LIN {X 0,Y 467.594,Z 791.05,A -85,B 0,C 180,E1 -7505.746,E2 -7505.746} C_VEL
LIN {X 0,Y 467.216,Z 798.675,A -85,B 0,C 180,E1 -7507.133,E2 -7507.133} C_VEL
LIN {X 0,Y 467.007,Z 804.577,A -85,B 0,C 180,E1 -7508.506,E2 -7508.506} C_VEL
LIN {X 0,Y 466.843,Z 809.072,A -85,B 0,C 180,E1 -7509.847,E2 -7509.847} C_VEL
LIN {X 0,Y 466.705,Z 813.073,A -85,B 0,C 180,E1 -7511.496,E2 -7511.496} C_VEL
LIN {X 0,Y 466.63,Z 814.936,A -85,B 0,C 180,E1 -7512.667,E2 -7512.667} C_VEL
LIN {X 0,Y 466.577,Z 816.084,A -85,B 0,C 180,E1 -7513.858,E2 -7513.858} C_VEL
LIN {X 0,Y 466.568,Z 816.491,A -85,B 0,C 180,E1 -7515.069,E2 -7515.069} C_VEL
LIN {X 0,Y 466.584,Z 816.072,A -85,B 0,C 180,E1 -7516.302,E2 -7516.302} C_VEL
LIN {X 0,Y 466.641,Z 814.812,A -85,B 0,C 180,E1 -7517.558,E2 -7517.558} C_VEL
LIN {X 0,Y 466.745,Z 812.646,A -85,B 0,C 180,E1 -7518.838,E2 -7518.838} C_VEL
LIN {X 0,Y 466.842,Z 809.444,A -85,B 0,C 180,E1 -7520.152,E2 -7520.152} C_VEL
LIN {X 0,Y 467.011,Z 805.061,A -85,B 0,C 180,E1 -7521.492,E2 -7521.492} C_VEL
LIN {X 0,Y 467.267,Z 798.57,A -85,B 0,C 180,E1 -7523.014,E2 -7523.014} C_VEL
LIN {X 0,Y 467.568,Z 791.804,A -85,B 0,C 180,E1 -7524.258,E2 -7524.258} C_VEL
LIN {X 0,Y 467.987,Z 783.664,A -85,B 0,C 180,E1 -7525.471,E2 -7525.471} C_VEL
LIN {X 0,Y 468.465,Z 774.171,A -85,B 0,C 180,E1 -7526.621,E2 -7526.621} C_VEL
LIN {X 0,Y 468.906,Z 764.185,A -85,B 0,C 180,E1 -7527.601,E2 -7527.601} C_VEL
LIN {X 0,Y 469.422,Z 752.274,A -85,B 0,C 180,E1 -7528.524,E2 -7528.524} C_VEL
LIN {X 0,Y 469.902,Z 740.221,A -85,B 0,C 180,E1 -7529.249,E2 -7529.249} C_VEL
LIN {X 0,Y 470.237,Z 727.327,A -85,B 0,C 180,E1 -7529.816,E2 -7529.816} C_VEL
LIN {X 0,Y 470.482,Z 714.641,A -85,B 0,C 180,E1 -7530.195,E2 -7530.195} C_VEL
LIN {X 0,Y 470.92,Z 673.673,A -85,B 0,C 180,E1 -7530.864,E2 -7530.864} C_VEL
LIN {X 0,Y 471.328,Z 620.727,A -85,B 0,C 180,E1 -7531.703,E2 -7531.703} C_VEL
LIN {X 0,Y 468.51,Z 607.159,A -85,B 0,C 180,E1 -7532.05,E2 -7532.05} C_VEL
LIN {X 0,Y 468.72,Z 598.189,A -85,B 0,C 180,E1 -7534.108,E2 -7534.108} C_VEL
LIN {X 0,Y 467.618,Z 592.238,A -85,B 0,C 180,E1 -7535.588,E2 -7535.588} C_VEL
LIN {X 0,Y 467.576,Z 592.244,A -85,B 0,C 180,E1 -7538.855,E2 -7538.855} C_VEL
LIN {X 0,Y 467.622,Z 592.234,A -85,B 0,C 180,E1 -7541.603,E2 -7541.603} C_VEL
LIN {X 0,Y 467.628,Z 592.236,A -85,B 0,C 180,E1 -7544.305,E2 -7544.305} C_VEL
LIN {X 0,Y 467.687,Z 592.225,A -85,B 0,C 180,E1 -7547.856,E2 -7547.856} C_VEL
LIN {X 0,Y 467.673,Z 592.229,A -85,B 0,C 180,E1 -7551.358,E2 -7551.358} C_VEL
LIN {X 0,Y 467.744,Z 592.218,A -85,B 0,C 180,E1 -7553.963,E2 -7553.963} C_VEL
LIN {X 0,Y 467.858,Z 592.205,A -85,B 0,C 180,E1 -7557.418,E2 -7557.418} C_VEL
LIN {X 0,Y 467.872,Z 592.201,A -85,B 0,C 180,E1 -7560,E2 -7560} C_VEL
LIN {X 0,Y 467.852,Z 592.207,A -85,B 0,C 180,E1 -7562.583,E2 -7562.583} C_VEL
LIN {X 0,Y 467.745,Z 592.216,A -85,B 0,C 180,E1 -7566.038,E2 -7566.038} C_VEL
LIN {X 0,Y 467.674,Z 592.23,A -85,B 0,C 180,E1 -7568.643,E2 -7568.643} C_VEL
LIN {X 0,Y 467.673,Z 592.225,A -85,B 0,C 180,E1 -7572.145,E2 -7572.145} C_VEL
LIN {X 0,Y 467.64,Z 592.227,A -85,B 0,C 180,E1 -7575.886,E2 -7575.886} C_VEL
LIN {X 0,Y 467.616,Z 592.237,A -85,B 0,C 180,E1 -7579.308,E2 -7579.308} C_VEL
LIN {X 0,Y 467.526,Z 592.242,A -85,B 0,C 180,E1 -7582.075,E2 -7582.075} C_VEL
LIN {X 0,Y 467.596,Z 592.239,A -85,B 0,C 180,E1 -7584.888,E2 -7584.888} C_VEL
LIN {X 0,Y 467.622,Z 592.232,A -85,B 0,C 180,E1 -7587.769,E2 -7587.769} C_VEL
LIN {X 0,Y 467.573,Z 592.242,A -85,B 0,C 180,E1 -7591.048,E2 -7591.048} C_VEL
LIN {X 0,Y 467.584,Z 592.235,A -85,B 0,C 180,E1 -7594.244,E2 -7594.244} C_VEL
LIN {X 0,Y 467.547,Z 592.247,A -85,B 0,C 180,E1 -7597.188,E2 -7597.188} C_VEL
LIN {X 0,Y 467.579,Z 592.236,A -85,B 0,C 180,E1 -7600.265,E2 -7600.265} C_VEL
LIN {X 0,Y 467.582,Z 592.238,A -85,B 0,C 180,E1 -7602.568,E2 -7602.568} C_VEL
LIN {X 0,Y 467.567,Z 592.243,A -85,B 0,C 180,E1 -7605.054,E2 -7605.054} C_VEL
LIN {X 0,Y 467.586,Z 592.244,A -85,B 0,C 180,E1 -7607.441,E2 -7607.441} C_VEL
LIN {X 0,Y 467.613,Z 592.235,A -85,B 0,C 180,E1 -7610.86,E2 -7610.86} C_VEL
LIN {X 0,Y 467.562,Z 592.242,A -85,B 0,C 180,E1 -7614.261,E2 -7614.261} C_VEL
LIN {X 0,Y 467.581,Z 592.244,A -85,B 0,C 180,E1 -7617.322,E2 -7617.322} C_VEL
LIN {X 0,Y 467.57,Z 592.242,A -85,B 0,C 180,E1 -7620.668,E2 -7620.668} C_VEL
LIN {X 0,Y 467.68,Z 592.255,A -85,B 0,C 180,E1 -7623.265,E2 -7623.265} C_VEL
LIN {X 0,Y 470.039,Z 604.523,A -85,B 0,C 180,E1 -7625.573,E2 -7625.573} C_VEL
LIN {X 0,Y 469.976,Z 610.728,A -85,B 0,C 180,E1 -7626.655,E2 -7626.655} C_VEL
LIN {X 0,Y 469.08,Z 629.475,A -85,B 0,C 180,E1 -7629.843,E2 -7629.843} C_VEL
LIN {X 0,Y 468.442,Z 645.546,A -85,B 0,C 180,E1 -7632.539,E2 -7632.539} C_VEL
LIN {X 0,Y 468.36,Z 648.312,A -85,B 0,C 180,E1 -7632.979,E2 -7632.979} C_VEL
LIN {X 0,Y 471.137,Z 667.101,A -85,B 0,C 180,E1 -7633.385,E2 -7633.385} C_VEL
LIN {X 0,Y 470.407,Z 757.136,A -85,B 0,C 180,E1 -7634.816,E2 -7634.816} C_VEL
LIN {X 0,Y 470.035,Z 770.301,A -85,B 0,C 180,E1 -7635.192,E2 -7635.192} C_VEL
LIN {X 0,Y 469.668,Z 782.454,A -85,B 0,C 180,E1 -7635.706,E2 -7635.706} C_VEL
LIN {X 0,Y 469.19,Z 793.935,A -85,B 0,C 180,E1 -7636.355,E2 -7636.355} C_VEL
LIN {X 0,Y 468.694,Z 805.881,A -85,B 0,C 180,E1 -7637.234,E2 -7637.234} C_VEL
LIN {X 0,Y 468.248,Z 816.36,A -85,B 0,C 180,E1 -7638.2,E2 -7638.2} C_VEL
LIN {X 0,Y 467.768,Z 825.036,A -85,B 0,C 180,E1 -7639.175,E2 -7639.175} C_VEL
LIN {X 0,Y 467.427,Z 833.045,A -85,B 0,C 180,E1 -7640.262,E2 -7640.262} C_VEL
LIN {X 0,Y 467.126,Z 840.876,A -85,B 0,C 180,E1 -7641.565,E2 -7641.565} C_VEL
LIN {X 0,Y 466.855,Z 848.078,A -85,B 0,C 180,E1 -7643.083,E2 -7643.083} C_VEL
LIN {X 0,Y 466.787,Z 852.882,A -85,B 0,C 180,E1 -7644.384,E2 -7644.384} C_VEL
LIN {X 0,Y 466.662,Z 856.552,A -85,B 0,C 180,E1 -7645.682,E2 -7645.682} C_VEL
LIN {X 0,Y 466.727,Z 858.454,A -85,B 0,C 180,E1 -7646.547,E2 -7646.547} C_VEL
LIN {X 0,Y 466.681,Z 859.877,A -85,B 0,C 180,E1 -7647.411,E2 -7647.411} C_VEL
LIN {X 0,Y 466.661,Z 860.895,A -85,B 0,C 180,E1 -7648.274,E2 -7648.274} C_VEL
LIN {X 0,Y 466.62,Z 861.518,A -85,B 0,C 180,E1 -7649.137,E2 -7649.137} C_VEL
LIN {X 0,Y 466.598,Z 861.745,A -85,B 0,C 180,E1 -7650,E2 -7650} C_VEL
LIN {X 0,Y 466.62,Z 861.534,A -85,B 0,C 180,E1 -7650.863,E2 -7650.863} C_VEL
LIN {X 0,Y 466.661,Z 860.929,A -85,B 0,C 180,E1 -7651.726,E2 -7651.726} C_VEL
LIN {X 0,Y 466.68,Z 859.93,A -85,B 0,C 180,E1 -7652.589,E2 -7652.589} C_VEL
LIN {X 0,Y 466.696,Z 858.521,A -85,B 0,C 180,E1 -7653.453,E2 -7653.453} C_VEL
LIN {X 0,Y 466.7,Z 855.559,A -85,B 0,C 180,E1 -7654.751,E2 -7654.751} C_VEL
LIN {X 0,Y 466.773,Z 851.546,A -85,B 0,C 180,E1 -7656.05,E2 -7656.05} C_VEL
LIN {X 0,Y 466.946,Z 845.366,A -85,B 0,C 180,E1 -7657.567,E2 -7657.567} C_VEL
LIN {X 0,Y 467.2,Z 838.62,A -85,B 0,C 180,E1 -7658.87,E2 -7658.87} C_VEL
LIN {X 0,Y 467.526,Z 830.248,A -85,B 0,C 180,E1 -7660.173,E2 -7660.173} C_VEL
LIN {X 0,Y 467.953,Z 821.64,A -85,B 0,C 180,E1 -7661.259,E2 -7661.259} C_VEL
LIN {X 0,Y 468.462,Z 811.469,A -85,B 0,C 180,E1 -7662.302,E2 -7662.302} C_VEL
LIN {X 0,Y 468.896,Z 800.495,A -85,B 0,C 180,E1 -7663.213,E2 -7663.213} C_VEL
LIN {X 0,Y 469.425,Z 788.908,A -85,B 0,C 180,E1 -7663.97,E2 -7663.97} C_VEL
LIN {X 0,Y 469.859,Z 776.886,A -85,B 0,C 180,E1 -7664.564,E2 -7664.564} C_VEL
LIN {X 0,Y 470.29,Z 763.907,A -85,B 0,C 180,E1 -7665.021,E2 -7665.021} C_VEL
LIN {X 0,Y 470.563,Z 750.082,A -85,B 0,C 180,E1 -7665.317,E2 -7665.317} C_VEL
LIN {X 0,Y 471.142,Z 667.137,A -85,B 0,C 180,E1 -7666.617,E2 -7666.617} C_VEL
LIN {X 0,Y 468.397,Z 648.688,A -85,B 0,C 180,E1 -7667.026,E2 -7667.026} C_VEL
LIN {X 0,Y 469.166,Z 630.051,A -85,B 0,C 180,E1 -7670.153,E2 -7670.153} C_VEL
LIN {X 0,Y 469.917,Z 613.979,A -85,B 0,C 180,E1 -7672.882,E2 -7672.882} C_VEL
LIN {X 0,Y 470.161,Z 604.995,A -85,B 0,C 180,E1 -7674.438,E2 -7674.438} C_VEL
LIN {X 0,Y 467.687,Z 592.23,A -85,B 0,C 180,E1 -7676.851,E2 -7676.851} C_VEL
LIN {X 0,Y 467.554,Z 592.244,A -85,B 0,C 180,E1 -7679.737,E2 -7679.737} C_VEL
LIN {X 0,Y 467.583,Z 592.241,A -85,B 0,C 180,E1 -7682.757,E2 -7682.757} C_VEL
LIN {X 0,Y 467.556,Z 592.24,A -85,B 0,C 180,E1 -7685.888,E2 -7685.888} C_VEL
LIN {X 0,Y 467.598,Z 592.235,A -85,B 0,C 180,E1 -7689.142,E2 -7689.142} C_VEL
LIN {X 0,Y 467.584,Z 592.244,A -85,B 0,C 180,E1 -7692.566,E2 -7692.566} C_VEL
LIN {X 0,Y 467.567,Z 592.241,A -85,B 0,C 180,E1 -7695.052,E2 -7695.052} C_VEL
LIN {X 0,Y 467.585,Z 592.236,A -85,B 0,C 180,E1 -7697.439,E2 -7697.439} C_VEL
LIN {X 0,Y 467.588,Z 592.242,A -85,B 0,C 180,E1 -7700.855,E2 -7700.855} C_VEL
LIN {X 0,Y 467.558,Z 592.241,A -85,B 0,C 180,E1 -7704.259,E2 -7704.259} C_VEL
LIN {X 0,Y 467.576,Z 592.239,A -85,B 0,C 180,E1 -7707.32,E2 -7707.32} C_VEL
LIN {X 0,Y 467.572,Z 592.242,A -85,B 0,C 180,E1 -7710.664,E2 -7710.664} C_VEL
LIN {X 0,Y 467.621,Z 592.236,A -85,B 0,C 180,E1 -7713.2,E2 -7713.2} C_VEL
LIN {X 0,Y 467.585,Z 592.237,A -85,B 0,C 180,E1 -7716.467,E2 -7716.467} C_VEL
LIN {X 0,Y 467.616,Z 592.232,A -85,B 0,C 180,E1 -7719.776,E2 -7719.776} C_VEL
LIN {X 0,Y 467.6,Z 592.235,A -85,B 0,C 180,E1 -7722.506,E2 -7722.506} C_VEL
LIN {X 0,Y 467.598,Z 592.243,A -85,B 0,C 180,E1 -7725.196,E2 -7725.196} C_VEL
LIN {X 0,Y 467.647,Z 592.229,A -85,B 0,C 180,E1 -7727.854,E2 -7727.854} C_VEL
LIN {X 0,Y 467.673,Z 592.232,A -85,B 0,C 180,E1 -7731.357,E2 -7731.357} C_VEL
LIN {X 0,Y 467.739,Z 592.217,A -85,B 0,C 180,E1 -7733.962,E2 -7733.962} C_VEL
LIN {X 0,Y 467.851,Z 592.211,A -85,B 0,C 180,E1 -7737.417,E2 -7737.417} C_VEL
LIN {X 0,Y 467.872,Z 592.201,A -85,B 0,C 180,E1 -7740,E2 -7740} C_VEL
LIN {X 0,Y 467.851,Z 592.202,A -85,B 0,C 180,E1 -7742.582,E2 -7742.582} C_VEL
LIN {X 0,Y 467.742,Z 592.218,A -85,B 0,C 180,E1 -7746.037,E2 -7746.037} C_VEL
LIN {X 0,Y 467.672,Z 592.224,A -85,B 0,C 180,E1 -7748.642,E2 -7748.642} C_VEL
LIN {X 0,Y 467.646,Z 592.23,A -85,B 0,C 180,E1 -7752.145,E2 -7752.145} C_VEL
LIN {X 0,Y 467.628,Z 592.238,A -85,B 0,C 180,E1 -7755.695,E2 -7755.695} C_VEL
LIN {X 0,Y 467.607,Z 592.233,A -85,B 0,C 180,E1 -7758.765,E2 -7758.765} C_VEL
LIN {X 0,Y 467.57,Z 592.239,A -85,B 0,C 180,E1 -7761.268,E2 -7761.268} C_VEL
LIN {X 0,Y 467.563,Z 592.246,A -85,B 0,C 180,E1 -7763.943,E2 -7763.943} C_VEL
LIN {X 0,Y 467.617,Z 592.231,A -85,B 0,C 180,E1 -7766.8,E2 -7766.8} C_VEL
LIN {X 0,Y 467.577,Z 592.241,A -85,B 0,C 180,E1 -7769.736,E2 -7769.736} C_VEL
LIN {X 0,Y 467.574,Z 592.237,A -85,B 0,C 180,E1 -7772.758,E2 -7772.758} C_VEL
LIN {X 0,Y 467.547,Z 592.246,A -85,B 0,C 180,E1 -7775.89,E2 -7775.89} C_VEL
LIN {X 0,Y 467.615,Z 592.232,A -85,B 0,C 180,E1 -7779.141,E2 -7779.141} C_VEL
LIN {X 0,Y 467.611,Z 592.236,A -85,B 0,C 180,E1 -7782.572,E2 -7782.572} C_VEL
LIN {X 0,Y 467.559,Z 592.246,A -85,B 0,C 180,E1 -7786.178,E2 -7786.178} C_VEL
LIN {X 0,Y 467.574,Z 592.24,A -85,B 0,C 180,E1 -7788.723,E2 -7788.723} C_VEL
LIN {X 0,Y 467.559,Z 592.241,A -85,B 0,C 180,E1 -7791.956,E2 -7791.956} C_VEL
LIN {X 0,Y 467.562,Z 592.239,A -85,B 0,C 180,E1 -7795.168,E2 -7795.168} C_VEL
LIN {X 0,Y 467.578,Z 592.241,A -85,B 0,C 180,E1 -7798.26,E2 -7798.26} C_VEL
LIN {X 0,Y 467.571,Z 592.238,A -85,B 0,C 180,E1 -7801.251,E2 -7801.251} C_VEL
LIN {X 0,Y 467.611,Z 592.234,A -85,B 0,C 180,E1 -7803.2,E2 -7803.2} C_VEL
LIN {X 0,Y 467.588,Z 592.241,A -85,B 0,C 180,E1 -7806.468,E2 -7806.468} C_VEL
LIN {X 0,Y 467.62,Z 592.231,A -85,B 0,C 180,E1 -7809.778,E2 -7809.778} C_VEL
LIN {X 0,Y 467.606,Z 592.238,A -85,B 0,C 180,E1 -7812.507,E2 -7812.507} C_VEL
LIN {X 0,Y 467.595,Z 592.235,A -85,B 0,C 180,E1 -7815.433,E2 -7815.433} C_VEL
LIN {X 0,Y 466.928,Z 592.319,A -85,B 0,C 180,E1 -7816.152,E2 -7816.152} C_VEL
LIN {X 0,Y 464.084,Z 592.674,A -85,B 0,C 180,E1 -7817.32,E2 -7817.32} C_VEL
LIN {X 0,Y 461.682,Z 592.972,A -85,B 0,C 180,E1 -7818.262,E2 -7818.262} C_VEL
LIN {X 0,Y 460.655,Z 593.106,A -85,B 0,C 180,E1 -7818.99,E2 -7818.99} C_VEL
LIN {X 0,Y 460.574,Z 593.11,A -85,B 0,C 180,E1 -7819.236,E2 -7819.236} C_VEL
LIN {X 0,Y 460.712,Z 593.095,A -85,B 0,C 180,E1 -7822.543,E2 -7822.543} C_VEL
LIN {X 0,Y 460.692,Z 593.099,A -85,B 0,C 180,E1 -7824.748,E2 -7824.748} C_VEL
LIN {X 0,Y 460.822,Z 593.082,A -85,B 0,C 180,E1 -7827.378,E2 -7827.378} C_VEL
LIN {X 0,Y 460.851,Z 593.074,A -85,B 0,C 180,E1 -7830,E2 -7830} C_VEL
LIN {X 0,Y 460.823,Z 593.08,A -85,B 0,C 180,E1 -7832.622,E2 -7832.622} C_VEL
LIN {X 0,Y 460.698,Z 593.093,A -85,B 0,C 180,E1 -7836.13,E2 -7836.13} C_VEL
LIN {X 0,Y 460.625,Z 593.105,A -85,B 0,C 180,E1 -7838.776,E2 -7838.776} C_VEL
LIN {X 0,Y 460.61,Z 593.104,A -85,B 0,C 180,E1 -7842.445,E2 -7842.445} C_VEL
LIN {X 0,Y 460.596,Z 593.107,A -85,B 0,C 180,E1 -7845.997,E2 -7845.997} C_VEL
LIN {X 0,Y 460.567,Z 593.112,A -85,B 0,C 180,E1 -7848.902,E2 -7848.902} C_VEL
LIN {X 0,Y 460.512,Z 593.125,A -85,B 0,C 180,E1 -7851.485,E2 -7851.485} C_VEL
LIN {X 0,Y 460.633,Z 593.212,A -85,B 0,C 180,E1 -7854.627,E2 -7854.627} C_VEL
LIN {X 0,Y 461.71,Z 599.757,A -85,B 0,C 180,E1 -7856.194,E2 -7856.194} C_VEL
LIN {X 0,Y 461.51,Z 606.979,A -85,B 0,C 180,E1 -7857.811,E2 -7857.811} C_VEL
LIN {X 0,Y 464.568,Z 622.378,A -85,B 0,C 180,E1 -7858.182,E2 -7858.182} C_VEL
LIN {X 0,Y 463.656,Z 713.559,A -85,B 0,C 180,E1 -7859.653,E2 -7859.653} C_VEL
LIN {X 0,Y 463.357,Z 727.425,A -85,B 0,C 180,E1 -7860.067,E2 -7860.067} C_VEL
LIN {X 0,Y 462.965,Z 740.325,A -85,B 0,C 180,E1 -7860.643,E2 -7860.643} C_VEL
LIN {X 0,Y 462.477,Z 752.601,A -85,B 0,C 180,E1 -7861.394,E2 -7861.394} C_VEL
LIN {X 0,Y 461.936,Z 764.155,A -85,B 0,C 180,E1 -7862.302,E2 -7862.302} C_VEL
LIN {X 0,Y 461.425,Z 774.936,A -85,B 0,C 180,E1 -7863.381,E2 -7863.381} C_VEL
LIN {X 0,Y 460.939,Z 784.574,A -85,B 0,C 180,E1 -7864.58,E2 -7864.58} C_VEL
LIN {X 0,Y 460.564,Z 792.034,A -85,B 0,C 180,E1 -7865.717,E2 -7865.717} C_VEL
LIN {X 0,Y 460.156,Z 799.828,A -85,B 0,C 180,E1 -7867.199,E2 -7867.199} C_VEL
LIN {X 0,Y 459.908,Z 806.333,A -85,B 0,C 180,E1 -7868.8,E2 -7868.8} C_VEL
LIN {X 0,Y 459.725,Z 810.475,A -85,B 0,C 180,E1 -7870.15,E2 -7870.15} C_VEL
LIN {X 0,Y 459.618,Z 813.471,A -85,B 0,C 180,E1 -7871.475,E2 -7871.475} C_VEL
LIN {X 0,Y 459.547,Z 815.452,A -85,B 0,C 180,E1 -7872.771,E2 -7872.771} C_VEL
LIN {X 0,Y 459.479,Z 816.535,A -85,B 0,C 180,E1 -7874.038,E2 -7874.038} C_VEL
LIN {X 0,Y 459.472,Z 816.802,A -85,B 0,C 180,E1 -7875.284,E2 -7875.284} C_VEL
LIN {X 0,Y 459.511,Z 816.299,A -85,B 0,C 180,E1 -7876.509,E2 -7876.509} C_VEL
LIN {X 0,Y 459.558,Z 815.019,A -85,B 0,C 180,E1 -7877.71,E2 -7877.71} C_VEL
LIN {X 0,Y 459.662,Z 813,A -85,B 0,C 180,E1 -7878.895,E2 -7878.895} C_VEL
LIN {X 0,Y 459.771,Z 810.274,A -85,B 0,C 180,E1 -7880.059,E2 -7880.059} C_VEL
LIN {X 0,Y 459.937,Z 805.782,A -85,B 0,C 180,E1 -7881.489,E2 -7881.489} C_VEL
LIN {X 0,Y 460.213,Z 799.458,A -85,B 0,C 180,E1 -7883.02,E2 -7883.02} C_VEL
LIN {X 0,Y 460.54,Z 792.863,A -85,B 0,C 180,E1 -7884.279,E2 -7884.279} C_VEL
LIN {X 0,Y 460.927,Z 785.531,A -85,B 0,C 180,E1 -7885.421,E2 -7885.421} C_VEL
LIN {X 0,Y 461.454,Z 776.05,A -85,B 0,C 180,E1 -7886.621,E2 -7886.621} C_VEL
LIN {X 0,Y 461.93,Z 765.542,A -85,B 0,C 180,E1 -7887.697,E2 -7887.697} C_VEL
LIN {X 0,Y 462.449,Z 754.398,A -85,B 0,C 180,E1 -7888.602,E2 -7888.602} C_VEL
LIN {X 0,Y 462.933,Z 742.386,A -85,B 0,C 180,E1 -7889.361,E2 -7889.361} C_VEL
LIN {X 0,Y 463.364,Z 729.575,A -85,B 0,C 180,E1 -7889.966,E2 -7889.966} C_VEL
LIN {X 0,Y 463.616,Z 716.872,A -85,B 0,C 180,E1 -7890.375,E2 -7890.375} C_VEL
LIN {X 0,Y 463.875,Z 697.07,A -85,B 0,C 180,E1 -7890.736,E2 -7890.736} C_VEL
LIN {X 0,Y 464.612,Z 621.891,A -85,B 0,C 180,E1 -7891.944,E2 -7891.944} C_VEL
LIN {X 0,Y 461.594,Z 607.587,A -85,B 0,C 180,E1 -7892.305,E2 -7892.305} C_VEL
LIN {X 0,Y 461.862,Z 600.852,A -85,B 0,C 180,E1 -7893.865,E2 -7893.865} C_VEL
LIN {X 0,Y 461.013,Z 595.306,A -85,B 0,C 180,E1 -7895.215,E2 -7895.215} C_VEL
LIN {X 0,Y 460.568,Z 593.117,A -85,B 0,C 180,E1 -7895.806,E2 -7895.806} C_VEL
LIN {X 0,Y 460.541,Z 593.116,A -85,B 0,C 180,E1 -7899.453,E2 -7899.453} C_VEL
LIN {X 0,Y 460.549,Z 593.118,A -85,B 0,C 180,E1 -7902.23,E2 -7902.23} C_VEL
LIN {X 0,Y 460.555,Z 593.118,A -85,B 0,C 180,E1 -7904.965,E2 -7904.965} C_VEL
LIN {X 0,Y 460.647,Z 593.102,A -85,B 0,C 180,E1 -7907.667,E2 -7907.667} C_VEL
LIN {X 0,Y 460.62,Z 593.108,A -85,B 0,C 180,E1 -7911.224,E2 -7911.224} C_VEL
LIN {X 0,Y 460.708,Z 593.094,A -85,B 0,C 180,E1 -7913.871,E2 -7913.871} C_VEL
LIN {X 0,Y 460.824,Z 593.081,A -85,B 0,C 180,E1 -7917.378,E2 -7917.378} C_VEL
LIN {X 0,Y 460.843,Z 593.077,A -85,B 0,C 180,E1 -7920,E2 -7920} C_VEL
LIN {X 0,Y 460.817,Z 593.084,A -85,B 0,C 180,E1 -7922.623,E2 -7922.623} C_VEL
LIN {X 0,Y 460.709,Z 593.093,A -85,B 0,C 180,E1 -7926.13,E2 -7926.13} C_VEL
LIN {X 0,Y 460.621,Z 593.11,A -85,B 0,C 180,E1 -7928.777,E2 -7928.777} C_VEL
LIN {X 0,Y 460.625,Z 593.105,A -85,B 0,C 180,E1 -7932.457,E2 -7932.457} C_VEL
LIN {X 0,Y 460.591,Z 593.105,A -85,B 0,C 180,E1 -7935.998,E2 -7935.998} C_VEL
LIN {X 0,Y 460.563,Z 593.116,A -85,B 0,C 180,E1 -7938.903,E2 -7938.903} C_VEL
LIN {X 0,Y 460.508,Z 593.12,A -85,B 0,C 180,E1 -7941.486,E2 -7941.486} C_VEL
LIN {X 0,Y 460.535,Z 593.115,A -85,B 0,C 180,E1 -7944.333,E2 -7944.333} C_VEL
LIN {X 0,Y 460.578,Z 593.116,A -85,B 0,C 180,E1 -7947.244,E2 -7947.244} C_VEL
LIN {X 0,Y 460.524,Z 593.115,A -85,B 0,C 180,E1 -7950.239,E2 -7950.239} C_VEL
LIN {X 0,Y 460.524,Z 593.121,A -85,B 0,C 180,E1 -7953.326,E2 -7953.326} C_VEL
LIN {X 0,Y 460.475,Z 593.122,A -85,B 0,C 180,E1 -7956.53,E2 -7956.53} C_VEL
LIN {X 0,Y 460.563,Z 593.113,A -85,B 0,C 180,E1 -7959.86,E2 -7959.86} C_VEL
LIN {X 0,Y 460.513,Z 593.12,A -85,B 0,C 180,E1 -7962.902,E2 -7962.902} C_VEL
LIN {X 0,Y 460.508,Z 593.123,A -85,B 0,C 180,E1 -7965.831,E2 -7965.831} C_VEL
LIN {X 0,Y 460.537,Z 593.117,A -85,B 0,C 180,E1 -7968.991,E2 -7968.991} C_VEL
LIN {X 0,Y 460.542,Z 593.12,A -85,B 0,C 180,E1 -7971.27,E2 -7971.27} C_VEL
LIN {X 0,Y 460.513,Z 593.119,A -85,B 0,C 180,E1 -7974.556,E2 -7974.556} C_VEL
LIN {X 0,Y 460.531,Z 593.124,A -85,B 0,C 180,E1 -7977.717,E2 -7977.717} C_VEL
LIN {X 0,Y 460.54,Z 593.118,A -85,B 0,C 180,E1 -7980.77,E2 -7980.77} C_VEL
LIN {X 0,Y 460.626,Z 593.217,A -85,B 0,C 180,E1 -7983.037,E2 -7983.037} C_VEL
LIN {X 0,Y 462.953,Z 605.027,A -85,B 0,C 180,E1 -7985.31,E2 -7985.31} C_VEL
LIN {X 0,Y 463.174,Z 609.126,A -85,B 0,C 180,E1 -7986.054,E2 -7986.054} C_VEL
LIN {X 0,Y 462.366,Z 625.149,A -85,B 0,C 180,E1 -7988.839,E2 -7988.839} C_VEL
LIN {X 0,Y 461.524,Z 643.862,A -85,B 0,C 180,E1 -7992.04,E2 -7992.04} C_VEL
LIN {X 0,Y 461.37,Z 647.878,A -85,B 0,C 180,E1 -7992.705,E2 -7992.705} C_VEL
LIN {X 0,Y 464.348,Z 668.691,A -85,B 0,C 180,E1 -7993.163,E2 -7993.163} C_VEL
LIN {X 0,Y 463.563,Z 756.607,A -85,B 0,C 180,E1 -7994.587,E2 -7994.587} C_VEL
LIN {X 0,Y 463.173,Z 769.816,A -85,B 0,C 180,E1 -7994.968,E2 -7994.968} C_VEL
LIN {X 0,Y 462.775,Z 781.997,A -85,B 0,C 180,E1 -7995.489,E2 -7995.489} C_VEL
LIN {X 0,Y 462.257,Z 793.501,A -85,B 0,C 180,E1 -7996.146,E2 -7996.146} C_VEL
LIN {X 0,Y 461.735,Z 805.465,A -85,B 0,C 180,E1 -7997.038,E2 -7997.038} C_VEL
LIN {X 0,Y 461.255,Z 815.957,A -85,B 0,C 180,E1 -7998.019,E2 -7998.019} C_VEL
LIN {X 0,Y 460.773,Z 824.645,A -85,B 0,C 180,E1 -7999.009,E2 -7999.009} C_VEL
LIN {X 0,Y 460.371,Z 832.661,A -85,B 0,C 180,E1 -8000.111,E2 -8000.111} C_VEL
LIN {X 0,Y 460.059,Z 840.503,A -85,B 0,C 180,E1 -8001.434,E2 -8001.434} C_VEL
LIN {X 0,Y 459.772,Z 847.713,A -85,B 0,C 180,E1 -8002.976,E2 -8002.976} C_VEL
LIN {X 0,Y 459.682,Z 852.522,A -85,B 0,C 180,E1 -8004.297,E2 -8004.297} C_VEL
LIN {X 0,Y 459.578,Z 856.198,A -85,B 0,C 180,E1 -8005.615,E2 -8005.615} C_VEL
LIN {X 0,Y 459.622,Z 858.102,A -85,B 0,C 180,E1 -8006.494,E2 -8006.494} C_VEL
LIN {X 0,Y 459.603,Z 859.529,A -85,B 0,C 180,E1 -8007.371,E2 -8007.371} C_VEL
LIN {X 0,Y 459.57,Z 860.548,A -85,B 0,C 180,E1 -8008.247,E2 -8008.247} C_VEL
LIN {X 0,Y 459.553,Z 861.174,A -85,B 0,C 180,E1 -8009.124,E2 -8009.124} C_VEL
LIN {X 0,Y 459.53,Z 861.402,A -85,B 0,C 180,E1 -8010,E2 -8010} C_VEL
LIN {X 0,Y 459.553,Z 861.192,A -85,B 0,C 180,E1 -8010.876,E2 -8010.876} C_VEL
LIN {X 0,Y 459.57,Z 860.586,A -85,B 0,C 180,E1 -8011.753,E2 -8011.753} C_VEL
LIN {X 0,Y 459.601,Z 859.586,A -85,B 0,C 180,E1 -8012.629,E2 -8012.629} C_VEL
LIN {X 0,Y 459.594,Z 858.174,A -85,B 0,C 180,E1 -8013.507,E2 -8013.507} C_VEL
LIN {X 0,Y 459.631,Z 855.21,A -85,B 0,C 180,E1 -8014.824,E2 -8014.824} C_VEL
LIN {X 0,Y 459.715,Z 850.142,A -85,B 0,C 180,E1 -8016.431,E2 -8016.431} C_VEL
LIN {X 0,Y 459.899,Z 843.98,A -85,B 0,C 180,E1 -8017.905,E2 -8017.905} C_VEL
LIN {X 0,Y 460.206,Z 836.994,A -85,B 0,C 180,E1 -8019.227,E2 -8019.227} C_VEL
LIN {X 0,Y 460.588,Z 828.233,A -85,B 0,C 180,E1 -8020.55,E2 -8020.55} C_VEL
LIN {X 0,Y 461.099,Z 819.266,A -85,B 0,C 180,E1 -8021.651,E2 -8021.651} C_VEL
LIN {X 0,Y 461.582,Z 808.4,A -85,B 0,C 180,E1 -8022.736,E2 -8022.736} C_VEL
LIN {X 0,Y 462.113,Z 796.987,A -85,B 0,C 180,E1 -8023.634,E2 -8023.634} C_VEL
LIN {X 0,Y 462.689,Z 784.431,A -85,B 0,C 180,E1 -8024.402,E2 -8024.402} C_VEL
LIN {X 0,Y 463.172,Z 771.595,A -85,B 0,C 180,E1 -8024.976,E2 -8024.976} C_VEL
LIN {X 0,Y 463.571,Z 757.947,A -85,B 0,C 180,E1 -8025.385,E2 -8025.385} C_VEL
LIN {X 0,Y 464.213,Z 684.288,A -85,B 0,C 180,E1 -8026.581,E2 -8026.581} C_VEL
LIN {X 0,Y 464.235,Z 667.208,A -85,B 0,C 180,E1 -8026.86,E2 -8026.86} C_VEL
LIN {X 0,Y 461.421,Z 648.364,A -85,B 0,C 180,E1 -8027.289,E2 -8027.289} C_VEL
LIN {X 0,Y 462.195,Z 631.06,A -85,B 0,C 180,E1 -8030.238,E2 -8030.238} C_VEL
LIN {X 0,Y 463.129,Z 612.34,A -85,B 0,C 180,E1 -8033.474,E2 -8033.474} C_VEL
LIN {X 0,Y 463.265,Z 606.741,A -85,B 0,C 180,E1 -8034.461,E2 -8034.461} C_VEL
LIN {X 0,Y 460.645,Z 593.107,A -85,B 0,C 180,E1 -8037.054,E2 -8037.054} C_VEL
LIN {X 0,Y 460.511,Z 593.124,A -85,B 0,C 180,E1 -8040.239,E2 -8040.239} C_VEL
LIN {X 0,Y 460.529,Z 593.114,A -85,B 0,C 180,E1 -8043.324,E2 -8043.324} C_VEL
LIN {X 0,Y 460.478,Z 593.129,A -85,B 0,C 180,E1 -8046.528,E2 -8046.528} C_VEL
LIN {X 0,Y 460.572,Z 593.11,A -85,B 0,C 180,E1 -8049.857,E2 -8049.857} C_VEL
LIN {X 0,Y 460.51,Z 593.121,A -85,B 0,C 180,E1 -8052.899,E2 -8052.899} C_VEL
LIN {X 0,Y 460.516,Z 593.116,A -85,B 0,C 180,E1 -8055.828,E2 -8055.828} C_VEL
LIN {X 0,Y 460.531,Z 593.119,A -85,B 0,C 180,E1 -8058.988,E2 -8058.988} C_VEL
LIN {X 0,Y 460.526,Z 593.117,A -85,B 0,C 180,E1 -8061.266,E2 -8061.266} C_VEL
LIN {X 0,Y 460.508,Z 593.122,A -85,B 0,C 180,E1 -8064.554,E2 -8064.554} C_VEL
LIN {X 0,Y 460.527,Z 593.115,A -85,B 0,C 180,E1 -8067.715,E2 -8067.715} C_VEL
LIN {X 0,Y 460.541,Z 593.119,A -85,B 0,C 180,E1 -8070.769,E2 -8070.769} C_VEL
LIN {X 0,Y 460.561,Z 593.111,A -85,B 0,C 180,E1 -8073.734,E2 -8073.734} C_VEL
LIN {X 0,Y 460.538,Z 593.116,A -85,B 0,C 180,E1 -8076.623,E2 -8076.623} C_VEL
LIN {X 0,Y 460.544,Z 593.116,A -85,B 0,C 180,E1 -8079.452,E2 -8079.452} C_VEL
LIN {X 0,Y 460.551,Z 593.112,A -85,B 0,C 180,E1 -8082.229,E2 -8082.229} C_VEL
LIN {X 0,Y 460.556,Z 593.116,A -85,B 0,C 180,E1 -8084.964,E2 -8084.964} C_VEL
LIN {X 0,Y 460.604,Z 593.106,A -85,B 0,C 180,E1 -8088.559,E2 -8088.559} C_VEL
LIN {X 0,Y 460.686,Z 593.095,A -85,B 0,C 180,E1 -8092.108,E2 -8092.108} C_VEL
LIN {X 0,Y 460.694,Z 593.095,A -85,B 0,C 180,E1 -8094.748,E2 -8094.748} C_VEL
LIN {X 0,Y 460.816,Z 593.087,A -85,B 0,C 180,E1 -8097.377,E2 -8097.377} C_VEL
LIN {X 0,Y 460.843,Z 593.077,A -85,B 0,C 180,E1 -8100,E2 -8100} C_VEL
LIN {X 0,Y 460.816,Z 593.079,A -85,B 0,C 180,E1 -8102.622,E2 -8102.622} C_VEL
LIN {X 0,Y 460.706,Z 593.094,A -85,B 0,C 180,E1 -8106.129,E2 -8106.129} C_VEL
LIN {X 0,Y 460.619,Z 593.103,A -85,B 0,C 180,E1 -8108.776,E2 -8108.776} C_VEL
LIN {X 0,Y 460.603,Z 593.106,A -85,B 0,C 180,E1 -8112.445,E2 -8112.445} C_VEL
LIN {X 0,Y 460.589,Z 593.112,A -85,B 0,C 180,E1 -8115.997,E2 -8115.997} C_VEL
LIN {X 0,Y 460.56,Z 593.11,A -85,B 0,C 180,E1 -8118.902,E2 -8118.902} C_VEL
LIN {X 0,Y 460.505,Z 593.121,A -85,B 0,C 180,E1 -8121.486,E2 -8121.486} C_VEL
LIN {X 0,Y 460.532,Z 593.117,A -85,B 0,C 180,E1 -8124.332,E2 -8124.332} C_VEL
LIN {X 0,Y 460.574,Z 593.109,A -85,B 0,C 180,E1 -8127.243,E2 -8127.243} C_VEL
LIN {X 0,Y 460.517,Z 593.121,A -85,B 0,C 180,E1 -8130.239,E2 -8130.239} C_VEL
LIN {X 0,Y 460.52,Z 593.116,A -85,B 0,C 180,E1 -8133.325,E2 -8133.325} C_VEL
LIN {X 0,Y 460.47,Z 593.125,A -85,B 0,C 180,E1 -8136.529,E2 -8136.529} C_VEL
LIN {X 0,Y 460.576,Z 593.113,A -85,B 0,C 180,E1 -8139.857,E2 -8139.857} C_VEL
LIN {X 0,Y 460.534,Z 593.115,A -85,B 0,C 180,E1 -8142.905,E2 -8142.905} C_VEL
LIN {X 0,Y 460.511,Z 593.119,A -85,B 0,C 180,E1 -8145.83,E2 -8145.83} C_VEL
LIN {X 0,Y 460.526,Z 593.116,A -85,B 0,C 180,E1 -8148.989,E2 -8148.989} C_VEL
LIN {X 0,Y 460.519,Z 593.116,A -85,B 0,C 180,E1 -8151.267,E2 -8151.267} C_VEL
LIN {X 0,Y 460.507,Z 593.124,A -85,B 0,C 180,E1 -8154.555,E2 -8154.555} C_VEL
LIN {X 0,Y 460.526,Z 593.115,A -85,B 0,C 180,E1 -8157.716,E2 -8157.716} C_VEL
LIN {X 0,Y 460.535,Z 593.119,A -85,B 0,C 180,E1 -8160.77,E2 -8160.77} C_VEL
LIN {X 0,Y 460.558,Z 593.111,A -85,B 0,C 180,E1 -8163.735,E2 -8163.735} C_VEL
LIN {X 0,Y 460.542,Z 593.121,A -85,B 0,C 180,E1 -8166.624,E2 -8166.624} C_VEL
LIN {X 0,Y 460.548,Z 593.113,A -85,B 0,C 180,E1 -8169.453,E2 -8169.453} C_VEL
LIN {X 0,Y 460.556,Z 593.113,A -85,B 0,C 180,E1 -8172.23,E2 -8172.23} C_VEL
LIN {X 0,Y 460.562,Z 593.117,A -85,B 0,C 180,E1 -8174.965,E2 -8174.965} C_VEL
LIN {X 0,Y 460.605,Z 593.105,A -85,B 0,C 180,E1 -8177.666,E2 -8177.666} C_VEL
LIN {X 0,Y 460.574,Z 593.11,A -85,B 0,C 180,E1 -8179.236,E2 -8179.236} C_VEL
LIN {X 0,Y 459.919,Z 593.194,A -85,B 0,C 180,E1 -8179.967,E2 -8179.967} C_VEL
LIN {X 0,Y 457.098,Z 593.552,A -85,B 0,C 180,E1 -8181.153,E2 -8181.153} C_VEL
LIN {X 0,Y 454.716,Z 593.85,A -85,B 0,C 180,E1 -8182.11,E2 -8182.11} C_VEL
LIN {X 0,Y 453.703,Z 593.972,A -85,B 0,C 180,E1 -8182.849,E2 -8182.849} C_VEL
LIN {X 0,Y 453.626,Z 593.979,A -85,B 0,C 180,E1 -8183.099,E2 -8183.099} C_VEL
LIN {X 0,Y 453.665,Z 593.974,A -85,B 0,C 180,E1 -8184.667,E2 -8184.667} C_VEL
LIN {X 0,Y 453.763,Z 593.962,A -85,B 0,C 180,E1 -8187.337,E2 -8187.337} C_VEL
LIN {X 0,Y 453.821,Z 593.95,A -85,B 0,C 180,E1 -8190,E2 -8190} C_VEL
LIN {X 0,Y 453.763,Z 593.96,A -85,B 0,C 180,E1 -8192.663,E2 -8192.663} C_VEL
LIN {X 0,Y 453.666,Z 593.969,A -85,B 0,C 180,E1 -8196.225,E2 -8196.225} C_VEL
LIN {X 0,Y 453.589,Z 593.983,A -85,B 0,C 180,E1 -8198.913,E2 -8198.913} C_VEL
LIN {X 0,Y 453.56,Z 593.983,A -85,B 0,C 180,E1 -8202.529,E2 -8202.529} C_VEL
LIN {X 0,Y 453.541,Z 593.985,A -85,B 0,C 180,E1 -8206.196,E2 -8206.196} C_VEL
LIN {X 0,Y 453.517,Z 593.991,A -85,B 0,C 180,E1 -8209.041,E2 -8209.041} C_VEL
LIN {X 0,Y 453.472,Z 593.998,A -85,B 0,C 180,E1 -8211.836,E2 -8211.836} C_VEL
LIN {X 0,Y 453.564,Z 594.049,A -85,B 0,C 180,E1 -8214.436,E2 -8214.436} C_VEL
LIN {X 0,Y 454.653,Z 600.378,A -85,B 0,C 180,E1 -8215.979,E2 -8215.979} C_VEL
LIN {X 0,Y 454.529,Z 607.138,A -85,B 0,C 180,E1 -8217.542,E2 -8217.542} C_VEL
LIN {X 0,Y 457.754,Z 622.922,A -85,B 0,C 180,E1 -8217.932,E2 -8217.932} C_VEL
LIN {X 0,Y 456.794,Z 713.802,A -85,B 0,C 180,E1 -8219.423,E2 -8219.423} C_VEL
LIN {X 0,Y 456.499,Z 727.374,A -85,B 0,C 180,E1 -8219.832,E2 -8219.832} C_VEL
LIN {X 0,Y 456.134,Z 739.388,A -85,B 0,C 180,E1 -8220.365,E2 -8220.365} C_VEL
LIN {X 0,Y 455.695,Z 749.846,A -85,B 0,C 180,E1 -8220.978,E2 -8220.978} C_VEL
LIN {X 0,Y 455.227,Z 760.741,A -85,B 0,C 180,E1 -8221.792,E2 -8221.792} C_VEL
LIN {X 0,Y 454.654,Z 771.056,A -85,B 0,C 180,E1 -8222.753,E2 -8222.753} C_VEL
LIN {X 0,Y 454.189,Z 780.61,A -85,B 0,C 180,E1 -8223.851,E2 -8223.851} C_VEL
LIN {X 0,Y 453.727,Z 788.579,A -85,B 0,C 180,E1 -8224.966,E2 -8224.966} C_VEL
LIN {X 0,Y 453.321,Z 796.241,A -85,B 0,C 180,E1 -8226.277,E2 -8226.277} C_VEL
LIN {X 0,Y 453.014,Z 802.848,A -85,B 0,C 180,E1 -8227.702,E2 -8227.702} C_VEL
LIN {X 0,Y 452.777,Z 807.932,A -85,B 0,C 180,E1 -8229.096,E2 -8229.096} C_VEL
LIN {X 0,Y 452.613,Z 812.322,A -85,B 0,C 180,E1 -8230.703,E2 -8230.703} C_VEL
LIN {X 0,Y 452.483,Z 814.621,A -85,B 0,C 180,E1 -8231.902,E2 -8231.902} C_VEL
LIN {X 0,Y 452.43,Z 816.196,A -85,B 0,C 180,E1 -8233.116,E2 -8233.116} C_VEL
LIN {X 0,Y 452.379,Z 817.058,A -85,B 0,C 180,E1 -8234.387,E2 -8234.387} C_VEL
LIN {X 0,Y 452.38,Z 817.089,A -85,B 0,C 180,E1 -8235.646,E2 -8235.646} C_VEL
LIN {X 0,Y 452.434,Z 816.329,A -85,B 0,C 180,E1 -8236.892,E2 -8236.892} C_VEL
LIN {X 0,Y 452.517,Z 814.7,A -85,B 0,C 180,E1 -8238.199,E2 -8238.199} C_VEL
LIN {X 0,Y 452.635,Z 812.111,A -85,B 0,C 180,E1 -8239.534,E2 -8239.534} C_VEL
LIN {X 0,Y 452.79,Z 808.42,A -85,B 0,C 180,E1 -8240.901,E2 -8240.901} C_VEL
LIN {X 0,Y 453.053,Z 802.49,A -85,B 0,C 180,E1 -8242.537,E2 -8242.537} C_VEL
LIN {X 0,Y 453.401,Z 795.997,A -85,B 0,C 180,E1 -8243.913,E2 -8243.913} C_VEL
LIN {X 0,Y 453.774,Z 788.629,A -85,B 0,C 180,E1 -8245.169,E2 -8245.169} C_VEL
LIN {X 0,Y 454.291,Z 779.526,A -85,B 0,C 180,E1 -8246.427,E2 -8246.427} C_VEL
LIN {X 0,Y 454.815,Z 770.05,A -85,B 0,C 180,E1 -8247.491,E2 -8247.491} C_VEL
LIN {X 0,Y 455.355,Z 759.081,A -85,B 0,C 180,E1 -8248.478,E2 -8248.478} C_VEL
LIN {X 0,Y 455.891,Z 747.615,A -85,B 0,C 180,E1 -8249.293,E2 -8249.293} C_VEL
LIN {X 0,Y 456.371,Z 735.221,A -85,B 0,C 180,E1 -8249.968,E2 -8249.968} C_VEL
LIN {X 0,Y 456.651,Z 721.892,A -85,B 0,C 180,E1 -8250.48,E2 -8250.48} C_VEL
LIN {X 0,Y 456.936,Z 709.473,A -85,B 0,C 180,E1 -8250.78,E2 -8250.78} C_VEL
LIN {X 0,Y 457.791,Z 622.33,A -85,B 0,C 180,E1 -8252.207,E2 -8252.207} C_VEL
LIN {X 0,Y 454.652,Z 607.94,A -85,B 0,C 180,E1 -8252.59,E2 -8252.59} C_VEL
LIN {X 0,Y 454.899,Z 601.899,A -85,B 0,C 180,E1 -8254.008,E2 -8254.008} C_VEL
LIN {X 0,Y 453.515,Z 593.997,A -85,B 0,C 180,E1 -8256.005,E2 -8256.005} C_VEL
LIN {X 0,Y 453.472,Z 593.999,A -85,B 0,C 180,E1 -8259.118,E2 -8259.118} C_VEL
LIN {X 0,Y 453.501,Z 593.994,A -85,B 0,C 180,E1 -8261.945,E2 -8261.945} C_VEL
LIN {X 0,Y 453.529,Z 593.995,A -85,B 0,C 180,E1 -8264.726,E2 -8264.726} C_VEL
LIN {X 0,Y 453.592,Z 593.981,A -85,B 0,C 180,E1 -8267.472,E2 -8267.472} C_VEL
LIN {X 0,Y 453.584,Z 593.987,A -85,B 0,C 180,E1 -8271.087,E2 -8271.087} C_VEL
LIN {X 0,Y 453.674,Z 593.971,A -85,B 0,C 180,E1 -8273.775,E2 -8273.775} C_VEL
LIN {X 0,Y 453.764,Z 593.961,A -85,B 0,C 180,E1 -8277.337,E2 -8277.337} C_VEL
LIN {X 0,Y 453.814,Z 593.953,A -85,B 0,C 180,E1 -8280,E2 -8280} C_VEL
LIN {X 0,Y 453.758,Z 593.964,A -85,B 0,C 180,E1 -8282.664,E2 -8282.664} C_VEL
LIN {X 0,Y 453.675,Z 593.97,A -85,B 0,C 180,E1 -8286.226,E2 -8286.226} C_VEL
LIN {X 0,Y 453.585,Z 593.987,A -85,B 0,C 180,E1 -8288.914,E2 -8288.914} C_VEL
LIN {X 0,Y 453.593,Z 593.981,A -85,B 0,C 180,E1 -8292.551,E2 -8292.551} C_VEL
LIN {X 0,Y 453.536,Z 593.983,A -85,B 0,C 180,E1 -8296.197,E2 -8296.197} C_VEL
LIN {X 0,Y 453.512,Z 593.994,A -85,B 0,C 180,E1 -8299.042,E2 -8299.042} C_VEL
LIN {X 0,Y 453.468,Z 593.994,A -85,B 0,C 180,E1 -8301.837,E2 -8301.837} C_VEL
LIN {X 0,Y 453.507,Z 593.993,A -85,B 0,C 180,E1 -8304.735,E2 -8304.735} C_VEL
LIN {X 0,Y 453.532,Z 593.986,A -85,B 0,C 180,E1 -8307.962,E2 -8307.962} C_VEL
LIN {X 0,Y 453.479,Z 593.994,A -85,B 0,C 180,E1 -8310.76,E2 -8310.76} C_VEL
LIN {X 0,Y 453.472,Z 593.994,A -85,B 0,C 180,E1 -8313.914,E2 -8313.914} C_VEL
LIN {X 0,Y 453.466,Z 594.001,A -85,B 0,C 180,E1 -8317.189,E2 -8317.189} C_VEL
LIN {X 0,Y 453.518,Z 593.996,A -85,B 0,C 180,E1 -8319.447,E2 -8319.447} C_VEL
LIN {X 0,Y 453.474,Z 593.997,A -85,B 0,C 180,E1 -8321.936,E2 -8321.936} C_VEL
LIN {X 0,Y 453.484,Z 593.999,A -85,B 0,C 180,E1 -8325.472,E2 -8325.472} C_VEL
LIN {X 0,Y 453.479,Z 593.996,A -85,B 0,C 180,E1 -8328.211,E2 -8328.211} C_VEL
LIN {X 0,Y 453.528,Z 593.989,A -85,B 0,C 180,E1 -8330.789,E2 -8330.789} C_VEL
LIN {X 0,Y 453.456,Z 594.002,A -85,B 0,C 180,E1 -8333.918,E2 -8333.918} C_VEL
LIN {X 0,Y 453.483,Z 594,A -85,B 0,C 180,E1 -8337.152,E2 -8337.152} C_VEL
LIN {X 0,Y 453.475,Z 593.998,A -85,B 0,C 180,E1 -8340.269,E2 -8340.269} C_VEL
LIN {X 0,Y 453.607,Z 594.18,A -85,B 0,C 180,E1 -8342.803,E2 -8342.803} C_VEL
LIN {X 0,Y 456,Z 606.326,A -85,B 0,C 180,E1 -8345.192,E2 -8345.192} C_VEL
LIN {X 0,Y 456.268,Z 610.208,A -85,B 0,C 180,E1 -8345.91,E2 -8345.91} C_VEL
LIN {X 0,Y 455.312,Z 627.525,A -85,B 0,C 180,E1 -8348.969,E2 -8348.969} C_VEL
LIN {X 0,Y 454.51,Z 644.884,A -85,B 0,C 180,E1 -8351.986,E2 -8351.986} C_VEL
LIN {X 0,Y 454.411,Z 647.406,A -85,B 0,C 180,E1 -8352.421,E2 -8352.421} C_VEL
LIN {X 0,Y 457.549,Z 669.615,A -85,B 0,C 180,E1 -8352.921,E2 -8352.921} C_VEL
LIN {X 0,Y 456.723,Z 756.235,A -85,B 0,C 180,E1 -8354.35,E2 -8354.35} C_VEL
LIN {X 0,Y 456.279,Z 769.418,A -85,B 0,C 180,E1 -8354.735,E2 -8354.735} C_VEL
LIN {X 0,Y 455.843,Z 782.713,A -85,B 0,C 180,E1 -8355.32,E2 -8355.32} C_VEL
LIN {X 0,Y 455.245,Z 794.701,A -85,B 0,C 180,E1 -8356.042,E2 -8356.042} C_VEL
LIN {X 0,Y 454.693,Z 807.036,A -85,B 0,C 180,E1 -8357.007,E2 -8357.007} C_VEL
LIN {X 0,Y 454.228,Z 816.634,A -85,B 0,C 180,E1 -8357.944,E2 -8357.944} C_VEL
LIN {X 0,Y 453.654,Z 825.979,A -85,B 0,C 180,E1 -8359.061,E2 -8359.061} C_VEL
LIN {X 0,Y 453.205,Z 835.072,A -85,B 0,C 180,E1 -8360.404,E2 -8360.404} C_VEL
LIN {X 0,Y 452.915,Z 842.403,A -85,B 0,C 180,E1 -8361.748,E2 -8361.748} C_VEL
LIN {X 0,Y 452.694,Z 847.35,A -85,B 0,C 180,E1 -8362.866,E2 -8362.866} C_VEL
LIN {X 0,Y 452.58,Z 852.165,A -85,B 0,C 180,E1 -8364.207,E2 -8364.207} C_VEL
LIN {X 0,Y 452.5,Z 855.847,A -85,B 0,C 180,E1 -8365.546,E2 -8365.546} C_VEL
LIN {X 0,Y 452.519,Z 857.753,A -85,B 0,C 180,E1 -8366.438,E2 -8366.438} C_VEL
LIN {X 0,Y 452.527,Z 859.182,A -85,B 0,C 180,E1 -8367.33,E2 -8367.33} C_VEL
LIN {X 0,Y 452.488,Z 860.832,A -85,B 0,C 180,E1 -8369.11,E2 -8369.11} C_VEL
LIN {X 0,Y 452.464,Z 861.059,A -85,B 0,C 180,E1 -8370,E2 -8370} C_VEL
LIN {X 0,Y 452.488,Z 860.848,A -85,B 0,C 180,E1 -8370.89,E2 -8370.89} C_VEL
LIN {X 0,Y 452.523,Z 859.24,A -85,B 0,C 180,E1 -8372.67,E2 -8372.67} C_VEL
LIN {X 0,Y 452.493,Z 857.824,A -85,B 0,C 180,E1 -8373.562,E2 -8373.562} C_VEL
LIN {X 0,Y 452.561,Z 854.857,A -85,B 0,C 180,E1 -8374.9,E2 -8374.9} C_VEL
LIN {X 0,Y 452.629,Z 850.202,A -85,B 0,C 180,E1 -8376.416,E2 -8376.416} C_VEL
LIN {X 0,Y 452.852,Z 843.61,A -85,B 0,C 180,E1 -8378.029,E2 -8378.029} C_VEL
LIN {X 0,Y 453.146,Z 836.612,A -85,B 0,C 180,E1 -8379.372,E2 -8379.372} C_VEL
LIN {X 0,Y 453.564,Z 827.836,A -85,B 0,C 180,E1 -8380.716,E2 -8380.716} C_VEL
LIN {X 0,Y 454.127,Z 818.856,A -85,B 0,C 180,E1 -8381.832,E2 -8381.832} C_VEL
LIN {X 0,Y 454.532,Z 809.673,A -85,B 0,C 180,E1 -8382.775,E2 -8382.775} C_VEL
LIN {X 0,Y 455.035,Z 799.6,A -85,B 0,C 180,E1 -8383.623,E2 -8383.623} C_VEL
LIN {X 0,Y 455.587,Z 787.922,A -85,B 0,C 180,E1 -8384.403,E2 -8384.403} C_VEL
LIN {X 0,Y 456.079,Z 775.805,A -85,B 0,C 180,E1 -8385.015,E2 -8385.015} C_VEL
LIN {X 0,Y 456.553,Z 762.677,A -85,B 0,C 180,E1 -8385.484,E2 -8385.484} C_VEL
LIN {X 0,Y 456.838,Z 750.107,A -85,B 0,C 180,E1 -8385.76,E2 -8385.76} C_VEL
LIN {X 0,Y 457.452,Z 668.219,A -85,B 0,C 180,E1 -8387.091,E2 -8387.091} C_VEL
LIN {X 0,Y 454.475,Z 647.983,A -85,B 0,C 180,E1 -8387.566,E2 -8387.566} C_VEL
LIN {X 0,Y 455.389,Z 628.051,A -85,B 0,C 180,E1 -8391.027,E2 -8391.027} C_VEL
LIN {X 0,Y 456.321,Z 610.671,A -85,B 0,C 180,E1 -8394.087,E2 -8394.087} C_VEL
LIN {X 0,Y 456.102,Z 606.643,A -85,B 0,C 180,E1 -8394.827,E2 -8394.827} C_VEL
LIN {X 0,Y 453.596,Z 593.985,A -85,B 0,C 180,E1 -8397.322,E2 -8397.322} C_VEL
LIN {X 0,Y 453.476,Z 593.999,A -85,B 0,C 180,E1 -8400.759,E2 -8400.759} C_VEL
LIN {X 0,Y 453.478,Z 593.995,A -85,B 0,C 180,E1 -8403.912,E2 -8403.912} C_VEL
LIN {X 0,Y 453.47,Z 593.995,A -85,B 0,C 180,E1 -8407.187,E2 -8407.187} C_VEL
LIN {X 0,Y 453.526,Z 593.987,A -85,B 0,C 180,E1 -8409.445,E2 -8409.445} C_VEL
LIN {X 0,Y 453.476,Z 593.994,A -85,B 0,C 180,E1 -8411.934,E2 -8411.934} C_VEL
LIN {X 0,Y 453.488,Z 593.992,A -85,B 0,C 180,E1 -8415.469,E2 -8415.469} C_VEL
LIN {X 0,Y 453.478,Z 593.995,A -85,B 0,C 180,E1 -8418.209,E2 -8418.209} C_VEL
LIN {X 0,Y 453.516,Z 593.996,A -85,B 0,C 180,E1 -8420.788,E2 -8420.788} C_VEL
LIN {X 0,Y 453.452,Z 593.996,A -85,B 0,C 180,E1 -8423.916,E2 -8423.916} C_VEL
LIN {X 0,Y 453.477,Z 593.997,A -85,B 0,C 180,E1 -8427.15,E2 -8427.15} C_VEL
LIN {X 0,Y 453.508,Z 593.99,A -85,B 0,C 180,E1 -8430.27,E2 -8430.27} C_VEL
LIN {X 0,Y 453.507,Z 593.993,A -85,B 0,C 180,E1 -8433.294,E2 -8433.294} C_VEL
LIN {X 0,Y 453.496,Z 593.991,A -85,B 0,C 180,E1 -8436.238,E2 -8436.238} C_VEL
LIN {X 0,Y 453.475,Z 594.001,A -85,B 0,C 180,E1 -8439.117,E2 -8439.117} C_VEL
LIN {X 0,Y 453.503,Z 593.99,A -85,B 0,C 180,E1 -8441.944,E2 -8441.944} C_VEL
LIN {X 0,Y 453.531,Z 593.989,A -85,B 0,C 180,E1 -8444.726,E2 -8444.726} C_VEL
LIN {X 0,Y 453.553,Z 593.984,A -85,B 0,C 180,E1 -8448.378,E2 -8448.378} C_VEL
LIN {X 0,Y 453.643,Z 593.973,A -85,B 0,C 180,E1 -8451.985,E2 -8451.985} C_VEL
LIN {X 0,Y 453.667,Z 593.97,A -85,B 0,C 180,E1 -8454.666,E2 -8454.666} C_VEL
LIN {X 0,Y 453.757,Z 593.966,A -85,B 0,C 180,E1 -8457.336,E2 -8457.336} C_VEL
LIN {X 0,Y 453.814,Z 593.953,A -85,B 0,C 180,E1 -8460,E2 -8460} C_VEL
LIN {X 0,Y 453.757,Z 593.958,A -85,B 0,C 180,E1 -8462.663,E2 -8462.663} C_VEL
LIN {X 0,Y 453.673,Z 593.969,A -85,B 0,C 180,E1 -8466.225,E2 -8466.225} C_VEL
LIN {X 0,Y 453.583,Z 593.98,A -85,B 0,C 180,E1 -8468.913,E2 -8468.913} C_VEL
LIN {X 0,Y 453.553,Z 593.984,A -85,B 0,C 180,E1 -8472.529,E2 -8472.529} C_VEL
LIN {X 0,Y 453.534,Z 593.988,A -85,B 0,C 180,E1 -8476.196,E2 -8476.196} C_VEL
LIN {X 0,Y 453.51,Z 593.989,A -85,B 0,C 180,E1 -8479.041,E2 -8479.041} C_VEL
LIN {X 0,Y 453.466,Z 594.003,A -85,B 0,C 180,E1 -8481.836,E2 -8481.836} C_VEL
LIN {X 0,Y 453.504,Z 593.99,A -85,B 0,C 180,E1 -8484.734,E2 -8484.734} C_VEL
LIN {X 0,Y 453.529,Z 593.995,A -85,B 0,C 180,E1 -8487.961,E2 -8487.961} C_VEL
LIN {X 0,Y 453.473,Z 593.994,A -85,B 0,C 180,E1 -8490.759,E2 -8490.759} C_VEL
LIN {X 0,Y 453.469,Z 594,A -85,B 0,C 180,E1 -8493.913,E2 -8493.913} C_VEL
LIN {X 0,Y 453.463,Z 593.995,A -85,B 0,C 180,E1 -8497.188,E2 -8497.188} C_VEL
LIN {X 0,Y 453.528,Z 593.987,A -85,B 0,C 180,E1 -8499.445,E2 -8499.445} C_VEL
LIN {X 0,Y 453.483,Z 593.992,A -85,B 0,C 180,E1 -8502.992,E2 -8502.992} C_VEL
LIN {X 0,Y 453.465,Z 593.997,A -85,B 0,C 180,E1 -8505.78,E2 -8505.78} C_VEL
LIN {X 0,Y 453.474,Z 594,A -85,B 0,C 180,E1 -8508.21,E2 -8508.21} C_VEL
LIN {X 0,Y 453.508,Z 593.992,A -85,B 0,C 180,E1 -8510.79,E2 -8510.79} C_VEL
LIN {X 0,Y 453.45,Z 593.998,A -85,B 0,C 180,E1 -8513.918,E2 -8513.918} C_VEL
LIN {X 0,Y 453.477,Z 593.994,A -85,B 0,C 180,E1 -8517.152,E2 -8517.152} C_VEL
LIN {X 0,Y 453.469,Z 593.998,A -85,B 0,C 180,E1 -8520.269,E2 -8520.269} C_VEL
LIN {X 0,Y 453.504,Z 593.99,A -85,B 0,C 180,E1 -8523.294,E2 -8523.294} C_VEL
LIN {X 0,Y 453.499,Z 593.993,A -85,B 0,C 180,E1 -8526.239,E2 -8526.239} C_VEL
LIN {X 0,Y 453.479,Z 593.996,A -85,B 0,C 180,E1 -8529.118,E2 -8529.118} C_VEL
LIN {X 0,Y 453.508,Z 593.989,A -85,B 0,C 180,E1 -8531.945,E2 -8531.945} C_VEL
LIN {X 0,Y 453.537,Z 593.993,A -85,B 0,C 180,E1 -8534.727,E2 -8534.727} C_VEL
LIN {X 0,Y 453.56,Z 593.984,A -85,B 0,C 180,E1 -8537.471,E2 -8537.471} C_VEL
LIN {X 0,Y 453.589,Z 593.985,A -85,B 0,C 180,E1 -8541.087,E2 -8541.087} C_VEL
LIN {X 0,Y 453.626,Z 593.979,A -85,B 0,C 180,E1 -8543.099,E2 -8543.099} C_VEL
LIN {X 0,Y 452.942,Z 594.062,A -85,B 0,C 180,E1 -8543.84,E2 -8543.84} C_VEL
LIN {X 0,Y 449.997,Z 594.434,A -85,B 0,C 180,E1 -8545.042,E2 -8545.042} C_VEL
LIN {X 0,Y 447.577,Z 594.731,A -85,B 0,C 180,E1 -8546.011,E2 -8546.011} C_VEL
LIN {X 0,Y 446.643,Z 594.849,A -85,B 0,C 180,E1 -8546.762,E2 -8546.762} C_VEL
LIN {X 0,Y 446.623,Z 594.849,A -85,B 0,C 180,E1 -8547.015,E2 -8547.015} C_VEL
LIN {X 0,Y 446.791,Z 594.826,A -85,B 0,C 180,E1 -8550,E2 -8550} C_VEL
LIN {X 0,Y 446.707,Z 594.839,A -85,B 0,C 180,E1 -8552.705,E2 -8552.705} C_VEL
LIN {X 0,Y 446.636,Z 594.845,A -85,B 0,C 180,E1 -8556.324,E2 -8556.324} C_VEL
LIN {X 0,Y 446.535,Z 594.863,A -85,B 0,C 180,E1 -8559.055,E2 -8559.055} C_VEL
LIN {X 0,Y 446.518,Z 594.861,A -85,B 0,C 180,E1 -8562.729,E2 -8562.729} C_VEL
LIN {X 0,Y 446.492,Z 594.863,A -85,B 0,C 180,E1 -8566.228,E2 -8566.228} C_VEL
LIN {X 0,Y 446.465,Z 594.873,A -85,B 0,C 180,E1 -8569.303,E2 -8569.303} C_VEL
LIN {X 0,Y 446.413,Z 594.876,A -85,B 0,C 180,E1 -8572.199,E2 -8572.199} C_VEL
LIN {X 0,Y 446.53,Z 595.036,A -85,B 0,C 180,E1 -8574.279,E2 -8574.279} C_VEL
LIN {X 0,Y 447.743,Z 602.296,A -85,B 0,C 180,E1 -8576.071,E2 -8576.071} C_VEL
LIN {X 0,Y 447.619,Z 607.605,A -85,B 0,C 180,E1 -8577.275,E2 -8577.275} C_VEL
LIN {X 0,Y 450.98,Z 624.574,A -85,B 0,C 180,E1 -8577.699,E2 -8577.699} C_VEL
LIN {X 0,Y 449.943,Z 714.352,A -85,B 0,C 180,E1 -8579.199,E2 -8579.199} C_VEL
LIN {X 0,Y 449.647,Z 727.99,A -85,B 0,C 180,E1 -8579.62,E2 -8579.62} C_VEL
LIN {X 0,Y 449.272,Z 739.362,A -85,B 0,C 180,E1 -8580.132,E2 -8580.132} C_VEL
LIN {X 0,Y 448.755,Z 751.555,A -85,B 0,C 180,E1 -8580.867,E2 -8580.867} C_VEL
LIN {X 0,Y 448.16,Z 763.28,A -85,B 0,C 180,E1 -8581.789,E2 -8581.789} C_VEL
LIN {X 0,Y 447.601,Z 773.526,A -85,B 0,C 180,E1 -8582.799,E2 -8582.799} C_VEL
LIN {X 0,Y 447.094,Z 783.331,A -85,B 0,C 180,E1 -8584.003,E2 -8584.003} C_VEL
LIN {X 0,Y 446.569,Z 791.973,A -85,B 0,C 180,E1 -8585.318,E2 -8585.318} C_VEL
LIN {X 0,Y 446.138,Z 799.624,A -85,B 0,C 180,E1 -8586.77,E2 -8586.77} C_VEL
LIN {X 0,Y 445.89,Z 804.78,A -85,B 0,C 180,E1 -8587.994,E2 -8587.994} C_VEL
LIN {X 0,Y 445.656,Z 809.488,A -85,B 0,C 180,E1 -8589.401,E2 -8589.401} C_VEL
LIN {X 0,Y 445.52,Z 812.983,A -85,B 0,C 180,E1 -8590.784,E2 -8590.784} C_VEL
LIN {X 0,Y 445.382,Z 815.399,A -85,B 0,C 180,E1 -8592.129,E2 -8592.129} C_VEL
LIN {X 0,Y 445.299,Z 817.204,A -85,B 0,C 180,E1 -8593.981,E2 -8593.981} C_VEL
LIN {X 0,Y 445.282,Z 817.499,A -85,B 0,C 180,E1 -8595.253,E2 -8595.253} C_VEL
LIN {X 0,Y 445.331,Z 817.002,A -85,B 0,C 180,E1 -8596.546,E2 -8596.546} C_VEL
LIN {X 0,Y 445.398,Z 815.629,A -85,B 0,C 180,E1 -8597.868,E2 -8597.868} C_VEL
LIN {X 0,Y 445.567,Z 812.229,A -85,B 0,C 180,E1 -8599.707,E2 -8599.707} C_VEL
LIN {X 0,Y 445.713,Z 809.079,A -85,B 0,C 180,E1 -8600.897,E2 -8600.897} C_VEL
LIN {X 0,Y 445.967,Z 804.008,A -85,B 0,C 180,E1 -8602.363,E2 -8602.363} C_VEL
LIN {X 0,Y 446.351,Z 797.089,A -85,B 0,C 180,E1 -8603.913,E2 -8603.913} C_VEL
LIN {X 0,Y 446.75,Z 789.755,A -85,B 0,C 180,E1 -8605.213,E2 -8605.213} C_VEL
LIN {X 0,Y 447.237,Z 781.582,A -85,B 0,C 180,E1 -8606.391,E2 -8606.391} C_VEL
LIN {X 0,Y 447.868,Z 771.02,A -85,B 0,C 180,E1 -8607.623,E2 -8607.623} C_VEL
LIN {X 0,Y 448.402,Z 760.671,A -85,B 0,C 180,E1 -8608.592,E2 -8608.592} C_VEL
LIN {X 0,Y 448.971,Z 749.465,A -85,B 0,C 180,E1 -8609.421,E2 -8609.421} C_VEL
LIN {X 0,Y 449.459,Z 737.518,A -85,B 0,C 180,E1 -8610.106,E2 -8610.106} C_VEL
LIN {X 0,Y 449.772,Z 724.354,A -85,B 0,C 180,E1 -8610.656,E2 -8610.656} C_VEL
LIN {X 0,Y 450.133,Z 711.047,A -85,B 0,C 180,E1 -8611.001,E2 -8611.001} C_VEL
LIN {X 0,Y 450.99,Z 623.191,A -85,B 0,C 180,E1 -8612.475,E2 -8612.475} C_VEL
LIN {X 0,Y 447.767,Z 608.272,A -85,B 0,C 180,E1 -8612.893,E2 -8612.893} C_VEL
LIN {X 0,Y 447.855,Z 601.847,A -85,B 0,C 180,E1 -8614.435,E2 -8614.435} C_VEL
LIN {X 0,Y 446.479,Z 594.873,A -85,B 0,C 180,E1 -8616.255,E2 -8616.255} C_VEL
LIN {X 0,Y 446.434,Z 594.874,A -85,B 0,C 180,E1 -8619.737,E2 -8619.737} C_VEL
LIN {X 0,Y 446.453,Z 594.876,A -85,B 0,C 180,E1 -8622.597,E2 -8622.597} C_VEL
LIN {X 0,Y 446.462,Z 594.87,A -85,B 0,C 180,E1 -8625.413,E2 -8625.413} C_VEL
LIN {X 0,Y 446.536,Z 594.862,A -85,B 0,C 180,E1 -8628.194,E2 -8628.194} C_VEL
LIN {X 0,Y 446.59,Z 594.854,A -85,B 0,C 180,E1 -8631.858,E2 -8631.858} C_VEL
LIN {X 0,Y 446.644,Z 594.85,A -85,B 0,C 180,E1 -8634.583,E2 -8634.583} C_VEL
LIN {X 0,Y 446.708,Z 594.841,A -85,B 0,C 180,E1 -8637.295,E2 -8637.295} C_VEL
LIN {X 0,Y 446.785,Z 594.829,A -85,B 0,C 180,E1 -8640,E2 -8640} C_VEL
LIN {X 0,Y 446.702,Z 594.843,A -85,B 0,C 180,E1 -8642.706,E2 -8642.706} C_VEL
LIN {X 0,Y 446.643,Z 594.846,A -85,B 0,C 180,E1 -8646.324,E2 -8646.324} C_VEL
LIN {X 0,Y 446.531,Z 594.863,A -85,B 0,C 180,E1 -8649.056,E2 -8649.056} C_VEL
LIN {X 0,Y 446.526,Z 594.863,A -85,B 0,C 180,E1 -8652.73,E2 -8652.73} C_VEL
LIN {X 0,Y 446.482,Z 594.863,A -85,B 0,C 180,E1 -8656.46,E2 -8656.46} C_VEL
LIN {X 0,Y 446.461,Z 594.871,A -85,B 0,C 180,E1 -8659.304,E2 -8659.304} C_VEL
LIN {X 0,Y 446.41,Z 594.872,A -85,B 0,C 180,E1 -8662.2,E2 -8662.2} C_VEL
LIN {X 0,Y 446.451,Z 594.873,A -85,B 0,C 180,E1 -8665.153,E2 -8665.153} C_VEL
LIN {X 0,Y 446.478,Z 594.864,A -85,B 0,C 180,E1 -8668.18,E2 -8668.18} C_VEL
LIN {X 0,Y 446.428,Z 594.875,A -85,B 0,C 180,E1 -8671.3,E2 -8671.3} C_VEL
LIN {X 0,Y 446.425,Z 594.871,A -85,B 0,C 180,E1 -8674.524,E2 -8674.524} C_VEL
LIN {X 0,Y 446.428,Z 594.871,A -85,B 0,C 180,E1 -8678.083,E2 -8678.083} C_VEL
LIN {X 0,Y 446.439,Z 594.872,A -85,B 0,C 180,E1 -8680.921,E2 -8680.921} C_VEL
LIN {X 0,Y 446.419,Z 594.878,A -85,B 0,C 180,E1 -8683.844,E2 -8683.844} C_VEL
LIN {X 0,Y 446.396,Z 594.877,A -85,B 0,C 180,E1 -8686.404,E2 -8686.404} C_VEL
LIN {X 0,Y 446.466,Z 594.872,A -85,B 0,C 180,E1 -8689.806,E2 -8689.806} C_VEL
LIN {X 0,Y 446.432,Z 594.875,A -85,B 0,C 180,E1 -8692.125,E2 -8692.125} C_VEL
LIN {X 0,Y 446.43,Z 594.88,A -85,B 0,C 180,E1 -8695.478,E2 -8695.478} C_VEL
LIN {X 0,Y 446.416,Z 594.874,A -85,B 0,C 180,E1 -8698.701,E2 -8698.701} C_VEL
LIN {X 0,Y 446.516,Z 594.868,A -85,B 0,C 180,E1 -8702.335,E2 -8702.335} C_VEL
LIN {X 0,Y 446.554,Z 594.975,A -85,B 0,C 180,E1 -8702.528,E2 -8702.528} C_VEL
LIN {X 0,Y 448.737,Z 605.966,A -85,B 0,C 180,E1 -8704.737,E2 -8704.737} C_VEL
LIN {X 0,Y 449.412,Z 610.204,A -85,B 0,C 180,E1 -8705.564,E2 -8705.564} C_VEL
LIN {X 0,Y 448.443,Z 627.256,A -85,B 0,C 180,E1 -8708.632,E2 -8708.632} C_VEL
LIN {X 0,Y 447.509,Z 645.921,A -85,B 0,C 180,E1 -8711.935,E2 -8711.935} C_VEL
LIN {X 0,Y 447.459,Z 647.148,A -85,B 0,C 180,E1 -8712.131,E2 -8712.131} C_VEL
LIN {X 0,Y 450.776,Z 670.504,A -85,B 0,C 180,E1 -8712.673,E2 -8712.673} C_VEL
LIN {X 0,Y 449.891,Z 755.943,A -85,B 0,C 180,E1 -8714.106,E2 -8714.106} C_VEL
LIN {X 0,Y 449.439,Z 769.093,A -85,B 0,C 180,E1 -8714.497,E2 -8714.497} C_VEL
LIN {X 0,Y 448.956,Z 782.371,A -85,B 0,C 180,E1 -8715.09,E2 -8715.09} C_VEL
LIN {X 0,Y 448.341,Z 794.353,A -85,B 0,C 180,E1 -8715.823,E2 -8715.823} C_VEL
LIN {X 0,Y 447.712,Z 806.684,A -85,B 0,C 180,E1 -8716.8,E2 -8716.8} C_VEL
LIN {X 0,Y 447.239,Z 816.273,A -85,B 0,C 180,E1 -8717.752,E2 -8717.752} C_VEL
LIN {X 0,Y 446.663,Z 825.614,A -85,B 0,C 180,E1 -8718.887,E2 -8718.887} C_VEL
LIN {X 0,Y 446.173,Z 834.703,A -85,B 0,C 180,E1 -8720.251,E2 -8720.251} C_VEL
LIN {X 0,Y 445.852,Z 842.033,A -85,B 0,C 180,E1 -8721.616,E2 -8721.616} C_VEL
LIN {X 0,Y 445.616,Z 846.987,A -85,B 0,C 180,E1 -8722.752,E2 -8722.752} C_VEL
LIN {X 0,Y 445.493,Z 851.21,A -85,B 0,C 180,E1 -8723.928,E2 -8723.928} C_VEL
LIN {X 0,Y 445.425,Z 855.496,A -85,B 0,C 180,E1 -8725.475,E2 -8725.475} C_VEL
LIN {X 0,Y 445.418,Z 857.403,A -85,B 0,C 180,E1 -8726.382,E2 -8726.382} C_VEL
LIN {X 0,Y 445.452,Z 858.836,A -85,B 0,C 180,E1 -8727.287,E2 -8727.287} C_VEL
LIN {X 0,Y 445.395,Z 860.488,A -85,B 0,C 180,E1 -8729.096,E2 -8729.096} C_VEL
LIN {X 0,Y 445.4,Z 860.716,A -85,B 0,C 180,E1 -8730,E2 -8730} C_VEL
LIN {X 0,Y 445.395,Z 860.503,A -85,B 0,C 180,E1 -8730.904,E2 -8730.904} C_VEL
LIN {X 0,Y 445.447,Z 858.894,A -85,B 0,C 180,E1 -8732.713,E2 -8732.713} C_VEL
LIN {X 0,Y 445.394,Z 857.474,A -85,B 0,C 180,E1 -8733.619,E2 -8733.619} C_VEL
LIN {X 0,Y 445.492,Z 854.503,A -85,B 0,C 180,E1 -8734.978,E2 -8734.978} C_VEL
LIN {X 0,Y 445.561,Z 849.013,A -85,B 0,C 180,E1 -8736.748,E2 -8736.748} C_VEL
LIN {X 0,Y 445.793,Z 843.239,A -85,B 0,C 180,E1 -8738.157,E2 -8738.157} C_VEL
LIN {X 0,Y 446.087,Z 836.229,A -85,B 0,C 180,E1 -8739.522,E2 -8739.522} C_VEL
LIN {X 0,Y 446.554,Z 827.44,A -85,B 0,C 180,E1 -8740.886,E2 -8740.886} C_VEL
LIN {X 0,Y 447.208,Z 817.462,A -85,B 0,C 180,E1 -8742.133,E2 -8742.133} C_VEL
LIN {X 0,Y 447.631,Z 807.342,A -85,B 0,C 180,E1 -8743.157,E2 -8743.157} C_VEL
LIN {X 0,Y 448.24,Z 796.061,A -85,B 0,C 180,E1 -8744.065,E2 -8744.065} C_VEL
LIN {X 0,Y 448.914,Z 783.433,A -85,B 0,C 180,E1 -8744.854,E2 -8744.854} C_VEL
LIN {X 0,Y 449.389,Z 771.17,A -85,B 0,C 180,E1 -8745.418,E2 -8745.418} C_VEL
LIN {X 0,Y 449.823,Z 757.649,A -85,B 0,C 180,E1 -8745.838,E2 -8745.838} C_VEL
LIN {X 0,Y 450.377,Z 712.549,A -85,B 0,C 180,E1 -8746.604,E2 -8746.604} C_VEL
LIN {X 0,Y 450.625,Z 668.955,A -85,B 0,C 180,E1 -8747.333,E2 -8747.333} C_VEL
LIN {X 0,Y 447.486,Z 647.76,A -85,B 0,C 180,E1 -8747.828,E2 -8747.828} C_VEL
LIN {X 0,Y 448.429,Z 629.045,A -85,B 0,C 180,E1 -8751.128,E2 -8751.128} C_VEL
LIN {X 0,Y 449.401,Z 611.761,A -85,B 0,C 180,E1 -8754.221,E2 -8754.221} C_VEL
LIN {X 0,Y 449.11,Z 607.645,A -85,B 0,C 180,E1 -8754.993,E2 -8754.993} C_VEL
LIN {X 0,Y 446.539,Z 594.864,A -85,B 0,C 180,E1 -8757.537,E2 -8757.537} C_VEL
LIN {X 0,Y 446.427,Z 594.878,A -85,B 0,C 180,E1 -8760.249,E2 -8760.249} C_VEL
LIN {X 0,Y 446.445,Z 594.869,A -85,B 0,C 180,E1 -8763.453,E2 -8763.453} C_VEL
LIN {X 0,Y 446.408,Z 594.878,A -85,B 0,C 180,E1 -8766.744,E2 -8766.744} C_VEL
LIN {X 0,Y 446.487,Z 594.864,A -85,B 0,C 180,E1 -8769.529,E2 -8769.529} C_VEL
LIN {X 0,Y 446.427,Z 594.88,A -85,B 0,C 180,E1 -8772.604,E2 -8772.604} C_VEL
LIN {X 0,Y 446.452,Z 594.871,A -85,B 0,C 180,E1 -8775.102,E2 -8775.102} C_VEL
LIN {X 0,Y 446.431,Z 594.878,A -85,B 0,C 180,E1 -8778.609,E2 -8778.609} C_VEL
LIN {X 0,Y 446.46,Z 594.872,A -85,B 0,C 180,E1 -8780.974,E2 -8780.974} C_VEL
LIN {X 0,Y 446.416,Z 594.875,A -85,B 0,C 180,E1 -8784.373,E2 -8784.373} C_VEL
LIN {X 0,Y 446.424,Z 594.872,A -85,B 0,C 180,E1 -8787.638,E2 -8787.638} C_VEL
LIN {X 0,Y 446.463,Z 594.873,A -85,B 0,C 180,E1 -8790.791,E2 -8790.791} C_VEL
LIN {X 0,Y 446.471,Z 594.866,A -85,B 0,C 180,E1 -8793.848,E2 -8793.848} C_VEL
LIN {X 0,Y 446.421,Z 594.877,A -85,B 0,C 180,E1 -8796.822,E2 -8796.822} C_VEL
LIN {X 0,Y 446.437,Z 594.871,A -85,B 0,C 180,E1 -8799.736,E2 -8799.736} C_VEL
LIN {X 0,Y 446.455,Z 594.869,A -85,B 0,C 180,E1 -8802.596,E2 -8802.596} C_VEL
LIN {X 0,Y 446.461,Z 594.872,A -85,B 0,C 180,E1 -8805.412,E2 -8805.412} C_VEL
LIN {X 0,Y 446.51,Z 594.861,A -85,B 0,C 180,E1 -8808.192,E2 -8808.192} C_VEL
LIN {X 0,Y 446.591,Z 594.852,A -85,B 0,C 180,E1 -8811.857,E2 -8811.857} C_VEL
LIN {X 0,Y 446.641,Z 594.845,A -85,B 0,C 180,E1 -8814.582,E2 -8814.582} C_VEL
LIN {X 0,Y 446.701,Z 594.844,A -85,B 0,C 180,E1 -8817.294,E2 -8817.294} C_VEL
LIN {X 0,Y 446.784,Z 594.828,A -85,B 0,C 180,E1 -8820,E2 -8820} C_VEL
LIN {X 0,Y 446.701,Z 594.837,A -85,B 0,C 180,E1 -8822.705,E2 -8822.705} C_VEL
LIN {X 0,Y 446.641,Z 594.845,A -85,B 0,C 180,E1 -8826.323,E2 -8826.323} C_VEL
LIN {X 0,Y 446.529,Z 594.86,A -85,B 0,C 180,E1 -8829.055,E2 -8829.055} C_VEL
LIN {X 0,Y 446.511,Z 594.861,A -85,B 0,C 180,E1 -8832.73,E2 -8832.73} C_VEL
LIN {X 0,Y 446.486,Z 594.866,A -85,B 0,C 180,E1 -8836.228,E2 -8836.228} C_VEL
LIN {X 0,Y 446.459,Z 594.869,A -85,B 0,C 180,E1 -8839.303,E2 -8839.303} C_VEL
LIN {X 0,Y 446.407,Z 594.877,A -85,B 0,C 180,E1 -8842.2,E2 -8842.2} C_VEL
LIN {X 0,Y 446.448,Z 594.869,A -85,B 0,C 180,E1 -8845.152,E2 -8845.152} C_VEL
LIN {X 0,Y 446.475,Z 594.871,A -85,B 0,C 180,E1 -8848.179,E2 -8848.179} C_VEL
LIN {X 0,Y 446.41,Z 594.874,A -85,B 0,C 180,E1 -8851.3,E2 -8851.3} C_VEL
LIN {X 0,Y 446.421,Z 594.875,A -85,B 0,C 180,E1 -8854.523,E2 -8854.523} C_VEL
LIN {X 0,Y 446.431,Z 594.878,A -85,B 0,C 180,E1 -8858.084,E2 -8858.084} C_VEL
LIN {X 0,Y 446.439,Z 594.87,A -85,B 0,C 180,E1 -8860.921,E2 -8860.921} C_VEL
LIN {X 0,Y 446.45,Z 594.871,A -85,B 0,C 180,E1 -8863.839,E2 -8863.839} C_VEL
LIN {X 0,Y 446.413,Z 594.88,A -85,B 0,C 180,E1 -8866.401,E2 -8866.401} C_VEL
LIN {X 0,Y 446.444,Z 594.871,A -85,B 0,C 180,E1 -8869.803,E2 -8869.803} C_VEL
LIN {X 0,Y 446.421,Z 594.877,A -85,B 0,C 180,E1 -8872.124,E2 -8872.124} C_VEL
LIN {X 0,Y 446.424,Z 594.871,A -85,B 0,C 180,E1 -8875.478,E2 -8875.478} C_VEL
LIN {X 0,Y 446.411,Z 594.879,A -85,B 0,C 180,E1 -8878.7,E2 -8878.7} C_VEL
LIN {X 0,Y 446.479,Z 594.865,A -85,B 0,C 180,E1 -8881.822,E2 -8881.822} C_VEL
LIN {X 0,Y 446.453,Z 594.873,A -85,B 0,C 180,E1 -8884.848,E2 -8884.848} C_VEL
LIN {X 0,Y 446.444,Z 594.872,A -85,B 0,C 180,E1 -8888.245,E2 -8888.245} C_VEL
LIN {X 0,Y 446.454,Z 594.868,A -85,B 0,C 180,E1 -8891.65,E2 -8891.65} C_VEL
LIN {X 0,Y 446.504,Z 594.865,A -85,B 0,C 180,E1 -8894.48,E2 -8894.48} C_VEL
LIN {X 0,Y 446.512,Z 594.862,A -85,B 0,C 180,E1 -8897.384,E2 -8897.384} C_VEL
LIN {X 0,Y 446.535,Z 594.866,A -85,B 0,C 180,E1 -8900.945,E2 -8900.945} C_VEL
LIN {X 0,Y 446.636,Z 594.846,A -85,B 0,C 180,E1 -8903.676,E2 -8903.676} C_VEL
LIN {X 0,Y 446.623,Z 594.849,A -85,B 0,C 180,E1 -8907.015,E2 -8907.015} C_VEL
LIN {X 0,Y 446.106,Z 594.919,A -85,B 0,C 180,E1 -8907.768,E2 -8907.768} C_VEL
LIN {X 0,Y 443.288,Z 595.276,A -85,B 0,C 180,E1 -8908.991,E2 -8908.991} C_VEL
LIN {X 0,Y 440.801,Z 595.585,A -85,B 0,C 180,E1 -8909.978,E2 -8909.978} C_VEL
LIN {X 0,Y 439.712,Z 595.715,A -85,B 0,C 180,E1 -8910.741,E2 -8910.741} C_VEL
LIN {X 0,Y 439.619,Z 595.724,A -85,B 0,C 180,E1 -8911,E2 -8911} C_VEL
LIN {X 0,Y 439.654,Z 595.718,A -85,B 0,C 180,E1 -8912.749,E2 -8912.749} C_VEL
LIN {X 0,Y 439.608,Z 595.721,A -85,B 0,C 180,E1 -8916.425,E2 -8916.425} C_VEL
LIN {X 0,Y 439.497,Z 595.742,A -85,B 0,C 180,E1 -8919.201,E2 -8919.201} C_VEL
LIN {X 0,Y 439.462,Z 595.742,A -85,B 0,C 180,E1 -8922.937,E2 -8922.937} C_VEL
LIN {X 0,Y 439.444,Z 595.741,A -85,B 0,C 180,E1 -8926.349,E2 -8926.349} C_VEL
LIN {X 0,Y 439.399,Z 595.754,A -85,B 0,C 180,E1 -8929.626,E2 -8929.626} C_VEL
LIN {X 0,Y 439.362,Z 595.755,A -85,B 0,C 180,E1 -8932.575,E2 -8932.575} C_VEL
LIN {X 0,Y 439.474,Z 595.812,A -85,B 0,C 180,E1 -8934.068,E2 -8934.068} C_VEL
LIN {X 0,Y 440.777,Z 603.557,A -85,B 0,C 180,E1 -8936.006,E2 -8936.006} C_VEL
LIN {X 0,Y 440.667,Z 607.67,A -85,B 0,C 180,E1 -8936.979,E2 -8936.979} C_VEL
LIN {X 0,Y 444.182,Z 624.998,A -85,B 0,C 180,E1 -8937.438,E2 -8937.438} C_VEL
LIN {X 0,Y 443.094,Z 715.199,A -85,B 0,C 180,E1 -8938.977,E2 -8938.977} C_VEL
LIN {X 0,Y 442.77,Z 728.888,A -85,B 0,C 180,E1 -8939.412,E2 -8939.412} C_VEL
LIN {X 0,Y 442.372,Z 740.689,A -85,B 0,C 180,E1 -8939.963,E2 -8939.963} C_VEL
LIN {X 0,Y 441.823,Z 752.429,A -85,B 0,C 180,E1 -8940.697,E2 -8940.697} C_VEL
LIN {X 0,Y 441.248,Z 763.526,A -85,B 0,C 180,E1 -8941.587,E2 -8941.587} C_VEL
LIN {X 0,Y 440.622,Z 774.554,A -85,B 0,C 180,E1 -8942.696,E2 -8942.696} C_VEL
LIN {X 0,Y 440.049,Z 784.672,A -85,B 0,C 180,E1 -8943.985,E2 -8943.985} C_VEL
LIN {X 0,Y 439.504,Z 793.392,A -85,B 0,C 180,E1 -8945.361,E2 -8945.361} C_VEL
LIN {X 0,Y 439.056,Z 800.777,A -85,B 0,C 180,E1 -8946.837,E2 -8946.837} C_VEL
LIN {X 0,Y 438.782,Z 806.536,A -85,B 0,C 180,E1 -8948.295,E2 -8948.295} C_VEL
LIN {X 0,Y 438.538,Z 811.304,A -85,B 0,C 180,E1 -8949.868,E2 -8949.868} C_VEL
LIN {X 0,Y 438.412,Z 814.076,A -85,B 0,C 180,E1 -8951.112,E2 -8951.112} C_VEL
LIN {X 0,Y 438.285,Z 816.22,A -85,B 0,C 180,E1 -8952.472,E2 -8952.472} C_VEL
LIN {X 0,Y 438.223,Z 817.458,A -85,B 0,C 180,E1 -8953.807,E2 -8953.807} C_VEL
LIN {X 0,Y 438.196,Z 817.867,A -85,B 0,C 180,E1 -8955.115,E2 -8955.115} C_VEL
LIN {X 0,Y 438.245,Z 817.454,A -85,B 0,C 180,E1 -8956.404,E2 -8956.404} C_VEL
LIN {X 0,Y 438.295,Z 816.284,A -85,B 0,C 180,E1 -8957.666,E2 -8957.666} C_VEL
LIN {X 0,Y 438.48,Z 813.184,A -85,B 0,C 180,E1 -8959.524,E2 -8959.524} C_VEL
LIN {X 0,Y 438.649,Z 809.983,A -85,B 0,C 180,E1 -8960.812,E2 -8960.812} C_VEL
LIN {X 0,Y 438.85,Z 805.775,A -85,B 0,C 180,E1 -8962.113,E2 -8962.113} C_VEL
LIN {X 0,Y 439.141,Z 800.436,A -85,B 0,C 180,E1 -8963.43,E2 -8963.43} C_VEL
LIN {X 0,Y 439.565,Z 793.173,A -85,B 0,C 180,E1 -8964.86,E2 -8964.86} C_VEL
LIN {X 0,Y 440.066,Z 785.066,A -85,B 0,C 180,E1 -8966.143,E2 -8966.143} C_VEL
LIN {X 0,Y 440.662,Z 776.073,A -85,B 0,C 180,E1 -8967.305,E2 -8967.305} C_VEL
LIN {X 0,Y 441.283,Z 765.456,A -85,B 0,C 180,E1 -8968.414,E2 -8968.414} C_VEL
LIN {X 0,Y 441.862,Z 754.867,A -85,B 0,C 180,E1 -8969.295,E2 -8969.295} C_VEL
LIN {X 0,Y 442.453,Z 742.352,A -85,B 0,C 180,E1 -8970.109,E2 -8970.109} C_VEL
LIN {X 0,Y 442.92,Z 729.437,A -85,B 0,C 180,E1 -8970.725,E2 -8970.725} C_VEL
LIN {X 0,Y 443.173,Z 718.173,A -85,B 0,C 180,E1 -8971.101,E2 -8971.101} C_VEL
LIN {X 0,Y 443.485,Z 699.007,A -85,B 0,C 180,E1 -8971.472,E2 -8971.472} C_VEL
LIN {X 0,Y 444.277,Z 624.18,A -85,B 0,C 180,E1 -8972.748,E2 -8972.748} C_VEL
LIN {X 0,Y 440.86,Z 608.632,A -85,B 0,C 180,E1 -8973.198,E2 -8973.198} C_VEL
LIN {X 0,Y 440.919,Z 603.267,A -85,B 0,C 180,E1 -8974.51,E2 -8974.51} C_VEL
LIN {X 0,Y 439.416,Z 595.753,A -85,B 0,C 180,E1 -8976.494,E2 -8976.494} C_VEL
LIN {X 0,Y 439.378,Z 595.753,A -85,B 0,C 180,E1 -8979.397,E2 -8979.397} C_VEL
LIN {X 0,Y 439.421,Z 595.752,A -85,B 0,C 180,E1 -8982.31,E2 -8982.31} C_VEL
LIN {X 0,Y 439.439,Z 595.747,A -85,B 0,C 180,E1 -8985.174,E2 -8985.174} C_VEL
LIN {X 0,Y 439.502,Z 595.737,A -85,B 0,C 180,E1 -8988.002,E2 -8988.002} C_VEL
LIN {X 0,Y 439.538,Z 595.733,A -85,B 0,C 180,E1 -8991.727,E2 -8991.727} C_VEL
LIN {X 0,Y 439.619,Z 595.725,A -85,B 0,C 180,E1 -8994.496,E2 -8994.496} C_VEL
LIN {X 0,Y 439.627,Z 595.721,A -85,B 0,C 180,E1 -8998.168,E2 -8998.168} C_VEL
LIN {X 0,Y 439.755,Z 595.704,A -85,B 0,C 180,E1 -9000,E2 -9000} C_VEL
LIN {X 0,Y 439.649,Z 595.723,A -85,B 0,C 180,E1 -9002.749,E2 -9002.749} C_VEL
LIN {X 0,Y 439.614,Z 595.723,A -85,B 0,C 180,E1 -9006.426,E2 -9006.426} C_VEL
LIN {X 0,Y 439.493,Z 595.738,A -85,B 0,C 180,E1 -9009.202,E2 -9009.202} C_VEL
LIN {X 0,Y 439.495,Z 595.739,A -85,B 0,C 180,E1 -9012.727,E2 -9012.727} C_VEL
LIN {X 0,Y 439.439,Z 595.74,A -85,B 0,C 180,E1 -9016.349,E2 -9016.349} C_VEL
LIN {X 0,Y 439.395,Z 595.75,A -85,B 0,C 180,E1 -9019.627,E2 -9019.627} C_VEL
LIN {X 0,Y 439.357,Z 595.752,A -85,B 0,C 180,E1 -9022.576,E2 -9022.576} C_VEL
LIN {X 0,Y 439.399,Z 595.747,A -85,B 0,C 180,E1 -9025.586,E2 -9025.586} C_VEL
LIN {X 0,Y 439.419,Z 595.744,A -85,B 0,C 180,E1 -9028.674,E2 -9028.674} C_VEL
LIN {X 0,Y 439.379,Z 595.746,A -85,B 0,C 180,E1 -9032.034,E2 -9032.034} C_VEL
LIN {X 0,Y 439.391,Z 595.75,A -85,B 0,C 180,E1 -9035.342,E2 -9035.342} C_VEL
LIN {X 0,Y 439.388,Z 595.747,A -85,B 0,C 180,E1 -9038.595,E2 -9038.595} C_VEL
LIN {X 0,Y 439.394,Z 595.751,A -85,B 0,C 180,E1 -9041.259,E2 -9041.259} C_VEL
LIN {X 0,Y 439.402,Z 595.749,A -85,B 0,C 180,E1 -9044.73,E2 -9044.73} C_VEL
LIN {X 0,Y 439.395,Z 595.753,A -85,B 0,C 180,E1 -9047.797,E2 -9047.797} C_VEL
LIN {X 0,Y 439.449,Z 595.744,A -85,B 0,C 180,E1 -9050.231,E2 -9050.231} C_VEL
LIN {X 0,Y 439.376,Z 595.758,A -85,B 0,C 180,E1 -9053.714,E2 -9053.714} C_VEL
LIN {X 0,Y 439.372,Z 595.757,A -85,B 0,C 180,E1 -9057.055,E2 -9057.055} C_VEL
LIN {X 0,Y 439.382,Z 595.753,A -85,B 0,C 180,E1 -9060.275,E2 -9060.275} C_VEL
LIN {X 0,Y 439.483,Z 595.83,A -85,B 0,C 180,E1 -9062.253,E2 -9062.253} C_VEL
LIN {X 0,Y 441.763,Z 607.077,A -85,B 0,C 180,E1 -9064.562,E2 -9064.562} C_VEL
LIN {X 0,Y 442.425,Z 610.747,A -85,B 0,C 180,E1 -9065.295,E2 -9065.295} C_VEL
LIN {X 0,Y 441.993,Z 620.259,A -85,B 0,C 180,E1 -9067.058,E2 -9067.058} C_VEL
LIN {X 0,Y 440.801,Z 641.616,A -85,B 0,C 180,E1 -9070.923,E2 -9070.923} C_VEL
LIN {X 0,Y 440.499,Z 646.653,A -85,B 0,C 180,E1 -9071.824,E2 -9071.824} C_VEL
LIN {X 0,Y 444.008,Z 671.261,A -85,B 0,C 180,E1 -9072.409,E2 -9072.409} C_VEL
LIN {X 0,Y 443.069,Z 755.65,A -85,B 0,C 180,E1 -9073.855,E2 -9073.855} C_VEL
LIN {X 0,Y 442.567,Z 769.524,A -85,B 0,C 180,E1 -9074.279,E2 -9074.279} C_VEL
LIN {X 0,Y 442.055,Z 782.028,A -85,B 0,C 180,E1 -9074.851,E2 -9074.851} C_VEL
LIN {X 0,Y 441.435,Z 794.005,A -85,B 0,C 180,E1 -9075.596,E2 -9075.596} C_VEL
LIN {X 0,Y 440.819,Z 805.781,A -85,B 0,C 180,E1 -9076.54,E2 -9076.54} C_VEL
LIN {X 0,Y 440.225,Z 815.923,A -85,B 0,C 180,E1 -9077.554,E2 -9077.554} C_VEL
LIN {X 0,Y 439.671,Z 825.268,A -85,B 0,C 180,E1 -9078.708,E2 -9078.708} C_VEL
LIN {X 0,Y 439.136,Z 834.358,A -85,B 0,C 180,E1 -9080.094,E2 -9080.094} C_VEL
LIN {X 0,Y 438.802,Z 841.692,A -85,B 0,C 180,E1 -9081.48,E2 -9081.48} C_VEL
LIN {X 0,Y 438.539,Z 846.641,A -85,B 0,C 180,E1 -9082.634,E2 -9082.634} C_VEL
LIN {X 0,Y 438.393,Z 851.3,A -85,B 0,C 180,E1 -9083.968,E2 -9083.968} C_VEL
LIN {X 0,Y 438.355,Z 855.151,A -85,B 0,C 180,E1 -9085.402,E2 -9085.402} C_VEL
LIN {X 0,Y 438.319,Z 857.056,A -85,B 0,C 180,E1 -9086.323,E2 -9086.323} C_VEL
LIN {X 0,Y 438.378,Z 858.492,A -85,B 0,C 180,E1 -9087.243,E2 -9087.243} C_VEL
LIN {X 0,Y 438.306,Z 860.144,A -85,B 0,C 180,E1 -9089.081,E2 -9089.081} C_VEL
LIN {X 0,Y 438.308,Z 860.372,A -85,B 0,C 180,E1 -9090,E2 -9090} C_VEL
LIN {X 0,Y 438.306,Z 860.159,A -85,B 0,C 180,E1 -9090.919,E2 -9090.919} C_VEL
LIN {X 0,Y 438.373,Z 858.548,A -85,B 0,C 180,E1 -9092.757,E2 -9092.757} C_VEL
LIN {X 0,Y 438.297,Z 857.123,A -85,B 0,C 180,E1 -9093.677,E2 -9093.677} C_VEL
LIN {X 0,Y 438.422,Z 854.149,A -85,B 0,C 180,E1 -9095.058,E2 -9095.058} C_VEL
LIN {X 0,Y 438.449,Z 850.105,A -85,B 0,C 180,E1 -9096.442,E2 -9096.442} C_VEL
LIN {X 0,Y 438.687,Z 843.879,A -85,B 0,C 180,E1 -9098.058,E2 -9098.058} C_VEL
LIN {X 0,Y 438.988,Z 837.085,A -85,B 0,C 180,E1 -9099.445,E2 -9099.445} C_VEL
LIN {X 0,Y 439.437,Z 828.649,A -85,B 0,C 180,E1 -9100.831,E2 -9100.831} C_VEL
LIN {X 0,Y 440.014,Z 819.959,A -85,B 0,C 180,E1 -9101.984,E2 -9101.984} C_VEL
LIN {X 0,Y 440.584,Z 808.926,A -85,B 0,C 180,E1 -9103.17,E2 -9103.17} C_VEL
LIN {X 0,Y 441.182,Z 798.622,A -85,B 0,C 180,E1 -9104.059,E2 -9104.059} C_VEL
LIN {X 0,Y 441.829,Z 786.811,A -85,B 0,C 180,E1 -9104.862,E2 -9104.862} C_VEL
LIN {X 0,Y 442.393,Z 773.251,A -85,B 0,C 180,E1 -9105.55,E2 -9105.55} C_VEL
LIN {X 0,Y 442.91,Z 760.088,A -85,B 0,C 180,E1 -9106.003,E2 -9106.003} C_VEL
LIN {X 0,Y 443.225,Z 742.653,A -85,B 0,C 180,E1 -9106.347,E2 -9106.347} C_VEL
LIN {X 0,Y 443.895,Z 670.414,A -85,B 0,C 180,E1 -9107.561,E2 -9107.561} C_VEL
LIN {X 0,Y 440.526,Z 647.428,A -85,B 0,C 180,E1 -9108.112,E2 -9108.112} C_VEL
LIN {X 0,Y 441.439,Z 630.023,A -85,B 0,C 180,E1 -9111.234,E2 -9111.234} C_VEL
LIN {X 0,Y 442.499,Z 612.664,A -85,B 0,C 180,E1 -9114.389,E2 -9114.389} C_VEL
LIN {X 0,Y 441.823,Z 607.269,A -85,B 0,C 180,E1 -9115.434,E2 -9115.434} C_VEL
LIN {X 0,Y 439.477,Z 595.743,A -85,B 0,C 180,E1 -9117.777,E2 -9117.777} C_VEL
LIN {X 0,Y 439.361,Z 595.757,A -85,B 0,C 180,E1 -9120.788,E2 -9120.788} C_VEL
LIN {X 0,Y 439.388,Z 595.751,A -85,B 0,C 180,E1 -9124.043,E2 -9124.043} C_VEL
LIN {X 0,Y 439.362,Z 595.751,A -85,B 0,C 180,E1 -9127.433,E2 -9127.433} C_VEL
LIN {X 0,Y 439.424,Z 595.744,A -85,B 0,C 180,E1 -9129.852,E2 -9129.852} C_VEL
LIN {X 0,Y 439.38,Z 595.757,A -85,B 0,C 180,E1 -9132.626,E2 -9132.626} C_VEL
LIN {X 0,Y 439.402,Z 595.747,A -85,B 0,C 180,E1 -9135.27,E2 -9135.27} C_VEL
LIN {X 0,Y 439.394,Z 595.755,A -85,B 0,C 180,E1 -9138.741,E2 -9138.741} C_VEL
LIN {X 0,Y 439.383,Z 595.749,A -85,B 0,C 180,E1 -9141.605,E2 -9141.605} C_VEL
LIN {X 0,Y 439.396,Z 595.755,A -85,B 0,C 180,E1 -9144.843,E2 -9144.843} C_VEL
LIN {X 0,Y 439.384,Z 595.749,A -85,B 0,C 180,E1 -9148.14,E2 -9148.14} C_VEL
LIN {X 0,Y 439.419,Z 595.747,A -85,B 0,C 180,E1 -9151.326,E2 -9151.326} C_VEL
LIN {X 0,Y 439.398,Z 595.748,A -85,B 0,C 180,E1 -9154.414,E2 -9154.414} C_VEL
LIN {X 0,Y 439.357,Z 595.755,A -85,B 0,C 180,E1 -9157.424,E2 -9157.424} C_VEL
LIN {X 0,Y 439.434,Z 595.745,A -85,B 0,C 180,E1 -9160.662,E2 -9160.662} C_VEL
LIN {X 0,Y 439.454,Z 595.74,A -85,B 0,C 180,E1 -9164.224,E2 -9164.224} C_VEL
LIN {X 0,Y 439.476,Z 595.738,A -85,B 0,C 180,E1 -9168.001,E2 -9168.001} C_VEL
LIN {X 0,Y 439.539,Z 595.732,A -85,B 0,C 180,E1 -9171.726,E2 -9171.726} C_VEL
LIN {X 0,Y 439.616,Z 595.72,A -85,B 0,C 180,E1 -9174.495,E2 -9174.495} C_VEL
LIN {X 0,Y 439.626,Z 595.719,A -85,B 0,C 180,E1 -9178.167,E2 -9178.167} C_VEL
LIN {X 0,Y 439.755,Z 595.704,A -85,B 0,C 180,E1 -9180,E2 -9180} C_VEL
LIN {X 0,Y 439.648,Z 595.716,A -85,B 0,C 180,E1 -9182.748,E2 -9182.748} C_VEL
LIN {X 0,Y 439.612,Z 595.72,A -85,B 0,C 180,E1 -9186.425,E2 -9186.425} C_VEL
LIN {X 0,Y 439.491,Z 595.738,A -85,B 0,C 180,E1 -9189.201,E2 -9189.201} C_VEL
LIN {X 0,Y 439.455,Z 595.74,A -85,B 0,C 180,E1 -9192.937,E2 -9192.937} C_VEL
LIN {X 0,Y 439.437,Z 595.743,A -85,B 0,C 180,E1 -9196.349,E2 -9196.349} C_VEL
LIN {X 0,Y 439.392,Z 595.753,A -85,B 0,C 180,E1 -9199.626,E2 -9199.626} C_VEL
LIN {X 0,Y 439.354,Z 595.753,A -85,B 0,C 180,E1 -9202.575,E2 -9202.575} C_VEL
LIN {X 0,Y 439.396,Z 595.751,A -85,B 0,C 180,E1 -9205.585,E2 -9205.585} C_VEL
LIN {X 0,Y 439.415,Z 595.745,A -85,B 0,C 180,E1 -9208.673,E2 -9208.673} C_VEL
LIN {X 0,Y 439.373,Z 595.758,A -85,B 0,C 180,E1 -9212.033,E2 -9212.033} C_VEL
LIN {X 0,Y 439.387,Z 595.749,A -85,B 0,C 180,E1 -9215.341,E2 -9215.341} C_VEL
LIN {X 0,Y 439.392,Z 595.75,A -85,B 0,C 180,E1 -9218.593,E2 -9218.593} C_VEL
LIN {X 0,Y 439.397,Z 595.747,A -85,B 0,C 180,E1 -9221.26,E2 -9221.26} C_VEL
LIN {X 0,Y 439.403,Z 595.749,A -85,B 0,C 180,E1 -9224.728,E2 -9224.728} C_VEL
LIN {X 0,Y 439.39,Z 595.75,A -85,B 0,C 180,E1 -9227.796,E2 -9227.796} C_VEL
LIN {X 0,Y 439.429,Z 595.749,A -85,B 0,C 180,E1 -9230.229,E2 -9230.229} C_VEL
LIN {X 0,Y 439.37,Z 595.751,A -85,B 0,C 180,E1 -9233.714,E2 -9233.714} C_VEL
LIN {X 0,Y 439.366,Z 595.752,A -85,B 0,C 180,E1 -9237.054,E2 -9237.054} C_VEL
LIN {X 0,Y 439.377,Z 595.754,A -85,B 0,C 180,E1 -9240.275,E2 -9240.275} C_VEL
LIN {X 0,Y 439.424,Z 595.744,A -85,B 0,C 180,E1 -9243.397,E2 -9243.397} C_VEL
LIN {X 0,Y 439.383,Z 595.754,A -85,B 0,C 180,E1 -9246.43,E2 -9246.43} C_VEL
LIN {X 0,Y 439.384,Z 595.749,A -85,B 0,C 180,E1 -9249.397,E2 -9249.397} C_VEL
LIN {X 0,Y 439.428,Z 595.746,A -85,B 0,C 180,E1 -9252.31,E2 -9252.31} C_VEL
LIN {X 0,Y 439.446,Z 595.744,A -85,B 0,C 180,E1 -9255.174,E2 -9255.174} C_VEL
LIN {X 0,Y 439.48,Z 595.737,A -85,B 0,C 180,E1 -9258.002,E2 -9258.002} C_VEL
LIN {X 0,Y 439.545,Z 595.729,A -85,B 0,C 180,E1 -9261.726,E2 -9261.726} C_VEL
LIN {X 0,Y 439.614,Z 595.722,A -85,B 0,C 180,E1 -9264.496,E2 -9264.496} C_VEL
LIN {X 0,Y 439.633,Z 595.718,A -85,B 0,C 180,E1 -9268.168,E2 -9268.168} C_VEL
LIN {X 0,Y 439.761,Z 595.702,A -85,B 0,C 180,E1 -9270,E2 -9270} C_VEL
LIN {X 0,Y 439.619,Z 595.724,A -85,B 0,C 180,E1 -9271,E2 -9271} C_VEL
LIN {X 0,Y 438.904,Z 595.811,A -85,B 0,C 180,E1 -9271.764,E2 -9271.764} C_VEL
LIN {X 0,Y 435.927,Z 596.186,A -85,B 0,C 180,E1 -9273.003,E2 -9273.003} C_VEL
LIN {X 0,Y 433.475,Z 596.489,A -85,B 0,C 180,E1 -9274.004,E2 -9274.004} C_VEL
LIN {X 0,Y 432.501,Z 596.609,A -85,B 0,C 180,E1 -9274.778,E2 -9274.778} C_VEL
LIN {X 0,Y 432.463,Z 596.611,A -85,B 0,C 180,E1 -9275.04,E2 -9275.04} C_VEL
LIN {X 0,Y 432.557,Z 596.602,A -85,B 0,C 180,E1 -9277.653,E2 -9277.653} C_VEL
LIN {X 0,Y 432.39,Z 596.628,A -85,B 0,C 180,E1 -9281.247,E2 -9281.247} C_VEL
LIN {X 0,Y 432.372,Z 596.622,A -85,B 0,C 180,E1 -9284.112,E2 -9284.112} C_VEL
LIN {X 0,Y 432.393,Z 596.623,A -85,B 0,C 180,E1 -9287.011,E2 -9287.011} C_VEL
LIN {X 0,Y 432.335,Z 596.632,A -85,B 0,C 180,E1 -9289.96,E2 -9289.96} C_VEL
LIN {X 0,Y 432.372,Z 596.629,A -85,B 0,C 180,E1 -9293.467,E2 -9293.467} C_VEL
LIN {X 0,Y 432.434,Z 596.831,A -85,B 0,C 180,E1 -9293.909,E2 -9293.909} C_VEL
LIN {X 0,Y 433.829,Z 604.836,A -85,B 0,C 180,E1 -9295.937,E2 -9295.937} C_VEL
LIN {X 0,Y 433.76,Z 607.956,A -85,B 0,C 180,E1 -9296.686,E2 -9296.686} C_VEL
LIN {X 0,Y 437.408,Z 626.391,A -85,B 0,C 180,E1 -9297.188,E2 -9297.188} C_VEL
LIN {X 0,Y 436.294,Z 714.781,A -85,B 0,C 180,E1 -9298.716,E2 -9298.716} C_VEL
LIN {X 0,Y 435.959,Z 727.837,A -85,B 0,C 180,E1 -9299.124,E2 -9299.124} C_VEL
LIN {X 0,Y 435.559,Z 740.007,A -85,B 0,C 180,E1 -9299.684,E2 -9299.684} C_VEL
LIN {X 0,Y 435.032,Z 750.489,A -85,B 0,C 180,E1 -9300.32,E2 -9300.32} C_VEL
LIN {X 0,Y 434.493,Z 761.479,A -85,B 0,C 180,E1 -9301.171,E2 -9301.171} C_VEL
LIN {X 0,Y 433.812,Z 771.884,A -85,B 0,C 180,E1 -9302.18,E2 -9302.18} C_VEL
LIN {X 0,Y 433.323,Z 780.682,A -85,B 0,C 180,E1 -9303.226,E2 -9303.226} C_VEL
LIN {X 0,Y 432.807,Z 788.479,A -85,B 0,C 180,E1 -9304.341,E2 -9304.341} C_VEL
LIN {X 0,Y 432.287,Z 796.92,A -85,B 0,C 180,E1 -9305.822,E2 -9305.822} C_VEL
LIN {X 0,Y 431.919,Z 802.878,A -85,B 0,C 180,E1 -9307.127,E2 -9307.127} C_VEL
LIN {X 0,Y 431.671,Z 808.232,A -85,B 0,C 180,E1 -9308.604,E2 -9308.604} C_VEL
LIN {X 0,Y 431.447,Z 812.242,A -85,B 0,C 180,E1 -9310.04,E2 -9310.04} C_VEL
LIN {X 0,Y 431.273,Z 815.125,A -85,B 0,C 180,E1 -9311.444,E2 -9311.444} C_VEL
LIN {X 0,Y 431.165,Z 817.36,A -85,B 0,C 180,E1 -9313.203,E2 -9313.203} C_VEL
LIN {X 0,Y 431.107,Z 818.115,A -85,B 0,C 180,E1 -9314.505,E2 -9314.505} C_VEL
LIN {X 0,Y 431.117,Z 818.097,A -85,B 0,C 180,E1 -9315.829,E2 -9315.829} C_VEL
LIN {X 0,Y 431.188,Z 817.225,A -85,B 0,C 180,E1 -9317.176,E2 -9317.176} C_VEL
LIN {X 0,Y 431.277,Z 815.467,A -85,B 0,C 180,E1 -9318.555,E2 -9318.555} C_VEL
LIN {X 0,Y 431.45,Z 812.739,A -85,B 0,C 180,E1 -9319.958,E2 -9319.958} C_VEL
LIN {X 0,Y 431.682,Z 808.898,A -85,B 0,C 180,E1 -9321.393,E2 -9321.393} C_VEL
LIN {X 0,Y 431.973,Z 803.265,A -85,B 0,C 180,E1 -9322.989,E2 -9322.989} C_VEL
LIN {X 0,Y 432.433,Z 795.76,A -85,B 0,C 180,E1 -9324.608,E2 -9324.608} C_VEL
LIN {X 0,Y 432.985,Z 787.34,A -85,B 0,C 180,E1 -9326.047,E2 -9326.047} C_VEL
LIN {X 0,Y 433.616,Z 778.468,A -85,B 0,C 180,E1 -9327.261,E2 -9327.261} C_VEL
LIN {X 0,Y 434.271,Z 768.168,A -85,B 0,C 180,E1 -9328.404,E2 -9328.404} C_VEL
LIN {X 0,Y 434.928,Z 756.924,A -85,B 0,C 180,E1 -9329.403,E2 -9329.403} C_VEL
LIN {X 0,Y 435.512,Z 744.919,A -85,B 0,C 180,E1 -9330.228,E2 -9330.228} C_VEL
LIN {X 0,Y 436.037,Z 732.655,A -85,B 0,C 180,E1 -9330.863,E2 -9330.863} C_VEL
LIN {X 0,Y 436.345,Z 720.252,A -85,B 0,C 180,E1 -9331.32,E2 -9331.32} C_VEL
LIN {X 0,Y 436.643,Z 706.444,A -85,B 0,C 180,E1 -9331.621,E2 -9331.621} C_VEL
LIN {X 0,Y 437.617,Z 625.588,A -85,B 0,C 180,E1 -9333.02,E2 -9333.02} C_VEL
LIN {X 0,Y 433.983,Z 609.156,A -85,B 0,C 180,E1 -9333.491,E2 -9333.491} C_VEL
LIN {X 0,Y 433.986,Z 604.708,A -85,B 0,C 180,E1 -9334.587,E2 -9334.587} C_VEL
LIN {X 0,Y 432.37,Z 596.631,A -85,B 0,C 180,E1 -9336.754,E2 -9336.754} C_VEL
LIN {X 0,Y 432.377,Z 596.63,A -85,B 0,C 180,E1 -9340.515,E2 -9340.515} C_VEL
LIN {X 0,Y 432.42,Z 596.62,A -85,B 0,C 180,E1 -9343.961,E2 -9343.961} C_VEL
LIN {X 0,Y 432.474,Z 596.612,A -85,B 0,C 180,E1 -9347.804,E2 -9347.804} C_VEL
LIN {X 0,Y 432.482,Z 596.612,A -85,B 0,C 180,E1 -9351.591,E2 -9351.591} C_VEL
LIN {X 0,Y 432.595,Z 596.6,A -85,B 0,C 180,E1 -9354.407,E2 -9354.407} C_VEL
LIN {X 0,Y 432.597,Z 596.597,A -85,B 0,C 180,E1 -9358.138,E2 -9358.138} C_VEL
LIN {X 0,Y 432.725,Z 596.58,A -85,B 0,C 180,E1 -9360,E2 -9360} C_VEL
LIN {X 0,Y 432.598,Z 596.602,A -85,B 0,C 180,E1 -9362.794,E2 -9362.794} C_VEL
LIN {X 0,Y 432.567,Z 596.602,A -85,B 0,C 180,E1 -9366.531,E2 -9366.531} C_VEL
LIN {X 0,Y 432.437,Z 596.616,A -85,B 0,C 180,E1 -9369.354,E2 -9369.354} C_VEL
LIN {X 0,Y 432.437,Z 596.618,A -85,B 0,C 180,E1 -9372.813,E2 -9372.813} C_VEL
LIN {X 0,Y 432.404,Z 596.617,A -85,B 0,C 180,E1 -9376.48,E2 -9376.48} C_VEL
LIN {X 0,Y 432.331,Z 596.628,A -85,B 0,C 180,E1 -9379.961,E2 -9379.961} C_VEL
LIN {X 0,Y 432.312,Z 596.632,A -85,B 0,C 180,E1 -9382.965,E2 -9382.965} C_VEL
LIN {X 0,Y 432.358,Z 596.622,A -85,B 0,C 180,E1 -9386.033,E2 -9386.033} C_VEL
LIN {X 0,Y 432.347,Z 596.627,A -85,B 0,C 180,E1 -9389.188,E2 -9389.188} C_VEL
LIN {X 0,Y 432.327,Z 596.624,A -85,B 0,C 180,E1 -9392.296,E2 -9392.296} C_VEL
LIN {X 0,Y 432.336,Z 596.627,A -85,B 0,C 180,E1 -9394.678,E2 -9394.678} C_VEL
LIN {X 0,Y 432.344,Z 596.625,A -85,B 0,C 180,E1 -9398.15,E2 -9398.15} C_VEL
LIN {X 0,Y 432.363,Z 596.63,A -85,B 0,C 180,E1 -9401.608,E2 -9401.608} C_VEL
LIN {X 0,Y 432.337,Z 596.629,A -85,B 0,C 180,E1 -9404.347,E2 -9404.347} C_VEL
LIN {X 0,Y 432.318,Z 596.634,A -85,B 0,C 180,E1 -9407.017,E2 -9407.017} C_VEL
LIN {X 0,Y 432.354,Z 596.63,A -85,B 0,C 180,E1 -9409.818,E2 -9409.818} C_VEL
LIN {X 0,Y 432.316,Z 596.634,A -85,B 0,C 180,E1 -9413.024,E2 -9413.024} C_VEL
LIN {X 0,Y 432.359,Z 596.632,A -85,B 0,C 180,E1 -9415.997,E2 -9415.997} C_VEL
LIN {X 0,Y 432.347,Z 596.633,A -85,B 0,C 180,E1 -9419.491,E2 -9419.491} C_VEL
LIN {X 0,Y 432.441,Z 596.781,A -85,B 0,C 180,E1 -9421.981,E2 -9421.981} C_VEL
LIN {X 0,Y 434.918,Z 608.845,A -85,B 0,C 180,E1 -9424.516,E2 -9424.516} C_VEL
LIN {X 0,Y 435.534,Z 613.517,A -85,B 0,C 180,E1 -9425.449,E2 -9425.449} C_VEL
LIN {X 0,Y 434.516,Z 629.384,A -85,B 0,C 180,E1 -9428.41,E2 -9428.41} C_VEL
LIN {X 0,Y 433.578,Z 646.26,A -85,B 0,C 180,E1 -9431.503,E2 -9431.503} C_VEL
LIN {X 0,Y 437.27,Z 671.683,A -85,B 0,C 180,E1 -9432.13,E2 -9432.13} C_VEL
LIN {X 0,Y 436.263,Z 755.525,A -85,B 0,C 180,E1 -9433.596,E2 -9433.596} C_VEL
LIN {X 0,Y 435.743,Z 769.289,A -85,B 0,C 180,E1 -9434.027,E2 -9434.027} C_VEL
LIN {X 0,Y 435.17,Z 781.73,A -85,B 0,C 180,E1 -9434.606,E2 -9434.606} C_VEL
LIN {X 0,Y 434.534,Z 793.672,A -85,B 0,C 180,E1 -9435.362,E2 -9435.362} C_VEL
LIN {X 0,Y 433.86,Z 805.663,A -85,B 0,C 180,E1 -9436.341,E2 -9436.341} C_VEL
LIN {X 0,Y 433.215,Z 815.573,A -85,B 0,C 180,E1 -9437.349,E2 -9437.349} C_VEL
LIN {X 0,Y 432.68,Z 824.92,A -85,B 0,C 180,E1 -9438.523,E2 -9438.523} C_VEL
LIN {X 0,Y 432.078,Z 834.014,A -85,B 0,C 180,E1 -9439.93,E2 -9439.93} C_VEL
LIN {X 0,Y 431.734,Z 841.35,A -85,B 0,C 180,E1 -9441.34,E2 -9441.34} C_VEL
LIN {X 0,Y 431.467,Z 846.302,A -85,B 0,C 180,E1 -9442.513,E2 -9442.513} C_VEL
LIN {X 0,Y 431.293,Z 851.399,A -85,B 0,C 180,E1 -9444.009,E2 -9444.009} C_VEL
LIN {X 0,Y 431.287,Z 854.813,A -85,B 0,C 180,E1 -9445.327,E2 -9445.327} C_VEL
LIN {X 0,Y 431.223,Z 856.717,A -85,B 0,C 180,E1 -9446.262,E2 -9446.262} C_VEL
LIN {X 0,Y 431.287,Z 858.151,A -85,B 0,C 180,E1 -9447.198,E2 -9447.198} C_VEL
LIN {X 0,Y 431.242,Z 859.173,A -85,B 0,C 180,E1 -9448.132,E2 -9448.132} C_VEL
LIN {X 0,Y 431.219,Z 859.802,A -85,B 0,C 180,E1 -9449.066,E2 -9449.066} C_VEL
LIN {X 0,Y 431.219,Z 860.027,A -85,B 0,C 180,E1 -9450,E2 -9450} C_VEL
LIN {X 0,Y 431.219,Z 859.81,A -85,B 0,C 180,E1 -9450.934,E2 -9450.934} C_VEL
LIN {X 0,Y 431.241,Z 859.199,A -85,B 0,C 180,E1 -9451.868,E2 -9451.868} C_VEL
LIN {X 0,Y 431.281,Z 858.192,A -85,B 0,C 180,E1 -9452.802,E2 -9452.802} C_VEL
LIN {X 0,Y 431.203,Z 856.76,A -85,B 0,C 180,E1 -9453.738,E2 -9453.738} C_VEL
LIN {X 0,Y 431.329,Z 853.777,A -85,B 0,C 180,E1 -9455.141,E2 -9455.141} C_VEL
LIN {X 0,Y 431.377,Z 849.723,A -85,B 0,C 180,E1 -9456.548,E2 -9456.548} C_VEL
LIN {X 0,Y 431.62,Z 843.479,A -85,B 0,C 180,E1 -9458.191,E2 -9458.191} C_VEL
LIN {X 0,Y 431.932,Z 836.668,A -85,B 0,C 180,E1 -9459.6,E2 -9459.6} C_VEL
LIN {X 0,Y 432.43,Z 828.209,A -85,B 0,C 180,E1 -9461.009,E2 -9461.009} C_VEL
LIN {X 0,Y 433.029,Z 819.491,A -85,B 0,C 180,E1 -9462.18,E2 -9462.18} C_VEL
LIN {X 0,Y 433.569,Z 809.446,A -85,B 0,C 180,E1 -9463.285,E2 -9463.285} C_VEL
LIN {X 0,Y 434.265,Z 798.09,A -85,B 0,C 180,E1 -9464.288,E2 -9464.288} C_VEL
LIN {X 0,Y 434.946,Z 786.201,A -85,B 0,C 180,E1 -9465.103,E2 -9465.103} C_VEL
LIN {X 0,Y 435.473,Z 773.858,A -85,B 0,C 180,E1 -9465.743,E2 -9465.743} C_VEL
LIN {X 0,Y 436.009,Z 761.274,A -85,B 0,C 180,E1 -9466.204,E2 -9466.204} C_VEL
LIN {X 0,Y 436.282,Z 748.355,A -85,B 0,C 180,E1 -9466.494,E2 -9466.494} C_VEL
LIN {X 0,Y 436.999,Z 670.516,A -85,B 0,C 180,E1 -9467.828,E2 -9467.828} C_VEL
LIN {X 0,Y 433.593,Z 647.062,A -85,B 0,C 180,E1 -9468.41,E2 -9468.41} C_VEL
LIN {X 0,Y 434.458,Z 630.991,A -85,B 0,C 180,E1 -9471.344,E2 -9471.344} C_VEL
LIN {X 0,Y 435.483,Z 614.967,A -85,B 0,C 180,E1 -9474.3,E2 -9474.3} C_VEL
LIN {X 0,Y 435.304,Z 610.825,A -85,B 0,C 180,E1 -9475.097,E2 -9475.097} C_VEL
LIN {X 0,Y 432.883,Z 598.744,A -85,B 0,C 180,E1 -9477.561,E2 -9477.561} C_VEL
LIN {X 0,Y 432.427,Z 596.622,A -85,B 0,C 180,E1 -9478.053,E2 -9478.053} C_VEL
LIN {X 0,Y 432.321,Z 596.632,A -85,B 0,C 180,E1 -9481.345,E2 -9481.345} C_VEL
LIN {X 0,Y 432.341,Z 596.631,A -85,B 0,C 180,E1 -9484.676,E2 -9484.676} C_VEL
LIN {X 0,Y 432.35,Z 596.628,A -85,B 0,C 180,E1 -9488.147,E2 -9488.147} C_VEL
LIN {X 0,Y 432.364,Z 596.623,A -85,B 0,C 180,E1 -9491.606,E2 -9491.606} C_VEL
LIN {X 0,Y 432.331,Z 596.631,A -85,B 0,C 180,E1 -9494.346,E2 -9494.346} C_VEL
LIN {X 0,Y 432.321,Z 596.632,A -85,B 0,C 180,E1 -9497.014,E2 -9497.014} C_VEL
LIN {X 0,Y 432.348,Z 596.625,A -85,B 0,C 180,E1 -9499.817,E2 -9499.817} C_VEL
LIN {X 0,Y 432.311,Z 596.635,A -85,B 0,C 180,E1 -9503.022,E2 -9503.022} C_VEL
LIN {X 0,Y 432.354,Z 596.624,A -85,B 0,C 180,E1 -9505.995,E2 -9505.995} C_VEL
LIN {X 0,Y 432.39,Z 596.62,A -85,B 0,C 180,E1 -9509.743,E2 -9509.743} C_VEL
LIN {X 0,Y 432.394,Z 596.622,A -85,B 0,C 180,E1 -9513.371,E2 -9513.371} C_VEL
LIN {X 0,Y 432.364,Z 596.623,A -85,B 0,C 180,E1 -9516.022,E2 -9516.022} C_VEL
LIN {X 0,Y 432.343,Z 596.634,A -85,B 0,C 180,E1 -9519.045,E2 -9519.045} C_VEL
LIN {X 0,Y 432.37,Z 596.622,A -85,B 0,C 180,E1 -9522.01,E2 -9522.01} C_VEL
LIN {X 0,Y 432.386,Z 596.625,A -85,B 0,C 180,E1 -9524.926,E2 -9524.926} C_VEL
LIN {X 0,Y 432.451,Z 596.614,A -85,B 0,C 180,E1 -9527.803,E2 -9527.803} C_VEL
LIN {X 0,Y 432.483,Z 596.612,A -85,B 0,C 180,E1 -9531.59,E2 -9531.59} C_VEL
LIN {X 0,Y 432.592,Z 596.595,A -85,B 0,C 180,E1 -9534.406,E2 -9534.406} C_VEL
LIN {X 0,Y 432.596,Z 596.595,A -85,B 0,C 180,E1 -9538.138,E2 -9538.138} C_VEL
LIN {X 0,Y 432.725,Z 596.58,A -85,B 0,C 180,E1 -9540,E2 -9540} C_VEL
LIN {X 0,Y 432.598,Z 596.595,A -85,B 0,C 180,E1 -9542.793,E2 -9542.793} C_VEL
LIN {X 0,Y 432.566,Z 596.598,A -85,B 0,C 180,E1 -9546.53,E2 -9546.53} C_VEL
LIN {X 0,Y 432.434,Z 596.619,A -85,B 0,C 180,E1 -9549.353,E2 -9549.353} C_VEL
LIN {X 0,Y 432.42,Z 596.616,A -85,B 0,C 180,E1 -9552.803,E2 -9552.803} C_VEL
LIN {X 0,Y 432.402,Z 596.619,A -85,B 0,C 180,E1 -9556.479,E2 -9556.479} C_VEL
LIN {X 0,Y 432.329,Z 596.634,A -85,B 0,C 180,E1 -9559.96,E2 -9559.96} C_VEL
LIN {X 0,Y 432.309,Z 596.63,A -85,B 0,C 180,E1 -9562.964,E2 -9562.964} C_VEL
LIN {X 0,Y 432.355,Z 596.631,A -85,B 0,C 180,E1 -9566.032,E2 -9566.032} C_VEL
LIN {X 0,Y 432.343,Z 596.626,A -85,B 0,C 180,E1 -9569.187,E2 -9569.187} C_VEL
LIN {X 0,Y 432.322,Z 596.633,A -85,B 0,C 180,E1 -9572.295,E2 -9572.295} C_VEL
LIN {X 0,Y 432.332,Z 596.628,A -85,B 0,C 180,E1 -9574.677,E2 -9574.677} C_VEL
LIN {X 0,Y 432.346,Z 596.634,A -85,B 0,C 180,E1 -9578.148,E2 -9578.148} C_VEL
LIN {X 0,Y 432.365,Z 596.624,A -85,B 0,C 180,E1 -9581.608,E2 -9581.608} C_VEL
LIN {X 0,Y 432.37,Z 596.629,A -85,B 0,C 180,E1 -9584.342,E2 -9584.342} C_VEL
LIN {X 0,Y 432.356,Z 596.631,A -85,B 0,C 180,E1 -9588.207,E2 -9588.207} C_VEL
LIN {X 0,Y 432.345,Z 596.625,A -85,B 0,C 180,E1 -9591.284,E2 -9591.284} C_VEL
LIN {X 0,Y 432.339,Z 596.633,A -85,B 0,C 180,E1 -9594.368,E2 -9594.368} C_VEL
LIN {X 0,Y 432.317,Z 596.629,A -85,B 0,C 180,E1 -9597.557,E2 -9597.557} C_VEL
LIN {X 0,Y 432.338,Z 596.631,A -85,B 0,C 180,E1 -9600.813,E2 -9600.813} C_VEL
LIN {X 0,Y 432.359,Z 596.625,A -85,B 0,C 180,E1 -9603.968,E2 -9603.968} C_VEL
LIN {X 0,Y 432.315,Z 596.632,A -85,B 0,C 180,E1 -9607.036,E2 -9607.036} C_VEL
LIN {X 0,Y 432.383,Z 596.626,A -85,B 0,C 180,E1 -9610.515,E2 -9610.515} C_VEL
LIN {X 0,Y 432.427,Z 596.615,A -85,B 0,C 180,E1 -9613.961,E2 -9613.961} C_VEL
LIN {X 0,Y 432.456,Z 596.612,A -85,B 0,C 180,E1 -9617.804,E2 -9617.804} C_VEL
LIN {X 0,Y 432.489,Z 596.608,A -85,B 0,C 180,E1 -9621.59,E2 -9621.59} C_VEL
LIN {X 0,Y 432.591,Z 596.596,A -85,B 0,C 180,E1 -9624.406,E2 -9624.406} C_VEL
LIN {X 0,Y 432.603,Z 596.593,A -85,B 0,C 180,E1 -9628.138,E2 -9628.138} C_VEL
LIN {X 0,Y 432.731,Z 596.577,A -85,B 0,C 180,E1 -9630,E2 -9630} C_VEL
LIN {X 0,Y 432.603,Z 596.597,A -85,B 0,C 180,E1 -9632.793,E2 -9632.793} C_VEL
LIN {X 0,Y 432.463,Z 596.611,A -85,B 0,C 180,E1 -9635.04,E2 -9635.04} C_VEL
LIN {X 0,Y 431.901,Z 596.684,A -85,B 0,C 180,E1 -9635.819,E2 -9635.819} C_VEL
LIN {X 0,Y 429.054,Z 597.042,A -85,B 0,C 180,E1 -9637.083,E2 -9637.083} C_VEL
LIN {X 0,Y 426.57,Z 597.347,A -85,B 0,C 180,E1 -9638.103,E2 -9638.103} C_VEL
LIN {X 0,Y 425.49,Z 597.483,A -85,B 0,C 180,E1 -9638.893,E2 -9638.893} C_VEL
LIN {X 0,Y 425.399,Z 597.492,A -85,B 0,C 180,E1 -9639.161,E2 -9639.161} C_VEL
LIN {X 0,Y 425.39,Z 597.495,A -85,B 0,C 180,E1 -9642.904,E2 -9642.904} C_VEL
LIN {X 0,Y 425.358,Z 597.496,A -85,B 0,C 180,E1 -9646.605,E2 -9646.605} C_VEL
LIN {X 0,Y 425.324,Z 597.507,A -85,B 0,C 180,E1 -9649.636,E2 -9649.636} C_VEL
LIN {X 0,Y 425.339,Z 597.505,A -85,B 0,C 180,E1 -9653.363,E2 -9653.363} C_VEL
LIN {X 0,Y 425.36,Z 597.621,A -85,B 0,C 180,E1 -9653.684,E2 -9653.684} C_VEL
LIN {X 0,Y 426.857,Z 606.087,A -85,B 0,C 180,E1 -9655.868,E2 -9655.868} C_VEL
LIN {X 0,Y 426.785,Z 608.263,A -85,B 0,C 180,E1 -9656.398,E2 -9656.398} C_VEL
LIN {X 0,Y 430.564,Z 626.194,A -85,B 0,C 180,E1 -9656.898,E2 -9656.898} C_VEL
LIN {X 0,Y 429.421,Z 715.767,A -85,B 0,C 180,E1 -9658.484,E2 -9658.484} C_VEL
LIN {X 0,Y 429.079,Z 729.727,A -85,B 0,C 180,E1 -9658.943,E2 -9658.943} C_VEL
LIN {X 0,Y 428.599,Z 742.154,A -85,B 0,C 180,E1 -9659.55,E2 -9659.55} C_VEL
LIN {X 0,Y 428.016,Z 754.212,A -85,B 0,C 180,E1 -9660.346,E2 -9660.346} C_VEL
LIN {X 0,Y 427.336,Z 765.446,A -85,B 0,C 180,E1 -9661.292,E2 -9661.292} C_VEL
LIN {X 0,Y 426.702,Z 775.566,A -85,B 0,C 180,E1 -9662.363,E2 -9662.363} C_VEL
LIN {X 0,Y 426.069,Z 785.582,A -85,B 0,C 180,E1 -9663.685,E2 -9663.685} C_VEL
LIN {X 0,Y 425.473,Z 794.048,A -85,B 0,C 180,E1 -9665.068,E2 -9665.068} C_VEL
LIN {X 0,Y 425.017,Z 801.187,A -85,B 0,C 180,E1 -9666.532,E2 -9666.532} C_VEL
LIN {X 0,Y 424.757,Z 806.016,A -85,B 0,C 180,E1 -9667.748,E2 -9667.748} C_VEL
LIN {X 0,Y 424.503,Z 809.998,A -85,B 0,C 180,E1 -9668.984,E2 -9668.984} C_VEL
LIN {X 0,Y 424.319,Z 813.483,A -85,B 0,C 180,E1 -9670.369,E2 -9670.369} C_VEL
LIN {X 0,Y 424.142,Z 816.07,A -85,B 0,C 180,E1 -9671.786,E2 -9671.786} C_VEL
LIN {X 0,Y 424.076,Z 817.703,A -85,B 0,C 180,E1 -9673.182,E2 -9673.182} C_VEL
LIN {X 0,Y 424.014,Z 818.467,A -85,B 0,C 180,E1 -9674.544,E2 -9674.544} C_VEL
LIN {X 0,Y 424.027,Z 818.431,A -85,B 0,C 180,E1 -9675.884,E2 -9675.884} C_VEL
LIN {X 0,Y 424.099,Z 817.589,A -85,B 0,C 180,E1 -9677.201,E2 -9677.201} C_VEL
LIN {X 0,Y 424.189,Z 816.008,A -85,B 0,C 180,E1 -9678.493,E2 -9678.493} C_VEL
LIN {X 0,Y 424.347,Z 813.71,A -85,B 0,C 180,E1 -9679.766,E2 -9679.766} C_VEL
LIN {X 0,Y 424.556,Z 810.516,A -85,B 0,C 180,E1 -9681.078,E2 -9681.078} C_VEL
LIN {X 0,Y 424.821,Z 805.744,A -85,B 0,C 180,E1 -9682.567,E2 -9682.567} C_VEL
LIN {X 0,Y 425.237,Z 799.518,A -85,B 0,C 180,E1 -9684.078,E2 -9684.078} C_VEL
LIN {X 0,Y 425.789,Z 791.521,A -85,B 0,C 180,E1 -9685.616,E2 -9685.616} C_VEL
LIN {X 0,Y 426.453,Z 782.013,A -85,B 0,C 180,E1 -9687.055,E2 -9687.055} C_VEL
LIN {X 0,Y 427.124,Z 772.373,A -85,B 0,C 180,E1 -9688.229,E2 -9688.229} C_VEL
LIN {X 0,Y 427.785,Z 761.727,A -85,B 0,C 180,E1 -9689.276,E2 -9689.276} C_VEL
LIN {X 0,Y 428.508,Z 749.514,A -85,B 0,C 180,E1 -9690.211,E2 -9690.211} C_VEL
LIN {X 0,Y 429.065,Z 737.736,A -85,B 0,C 180,E1 -9690.905,E2 -9690.905} C_VEL
LIN {X 0,Y 429.391,Z 725.134,A -85,B 0,C 180,E1 -9691.447,E2 -9691.447} C_VEL
LIN {X 0,Y 429.779,Z 712.259,A -85,B 0,C 180,E1 -9691.797,E2 -9691.797} C_VEL
LIN {X 0,Y 430.93,Z 626.763,A -85,B 0,C 180,E1 -9693.311,E2 -9693.311} C_VEL
LIN {X 0,Y 427.119,Z 609.446,A -85,B 0,C 180,E1 -9693.838,E2 -9693.838} C_VEL
LIN {X 0,Y 427.063,Z 606.161,A -85,B 0,C 180,E1 -9694.668,E2 -9694.668} C_VEL
LIN {X 0,Y 425.316,Z 597.508,A -85,B 0,C 180,E1 -9697.022,E2 -9697.022} C_VEL
LIN {X 0,Y 425.352,Z 597.504,A -85,B 0,C 180,E1 -9700.704,E2 -9700.704} C_VEL
LIN {X 0,Y 425.378,Z 597.496,A -85,B 0,C 180,E1 -9703.688,E2 -9703.688} C_VEL
LIN {X 0,Y 425.422,Z 597.491,A -85,B 0,C 180,E1 -9707.599,E2 -9707.599} C_VEL
LIN {X 0,Y 425.433,Z 597.491,A -85,B 0,C 180,E1 -9711.45,E2 -9711.45} C_VEL
LIN {X 0,Y 425.57,Z 597.474,A -85,B 0,C 180,E1 -9714.314,E2 -9714.314} C_VEL
LIN {X 0,Y 425.567,Z 597.472,A -85,B 0,C 180,E1 -9718.108,E2 -9718.108} C_VEL
LIN {X 0,Y 425.695,Z 597.456,A -85,B 0,C 180,E1 -9720,E2 -9720} C_VEL
LIN {X 0,Y 425.55,Z 597.48,A -85,B 0,C 180,E1 -9722.84,E2 -9722.84} C_VEL
LIN {X 0,Y 425.57,Z 597.471,A -85,B 0,C 180,E1 -9725.687,E2 -9725.687} C_VEL
LIN {X 0,Y 425.434,Z 597.491,A -85,B 0,C 180,E1 -9728.551,E2 -9728.551} C_VEL
LIN {X 0,Y 425.422,Z 597.49,A -85,B 0,C 180,E1 -9732.402,E2 -9732.402} C_VEL
LIN {X 0,Y 425.38,Z 597.491,A -85,B 0,C 180,E1 -9736.313,E2 -9736.313} C_VEL
LIN {X 0,Y 425.321,Z 597.503,A -85,B 0,C 180,E1 -9739.636,E2 -9739.636} C_VEL
LIN {X 0,Y 425.3,Z 597.509,A -85,B 0,C 180,E1 -9743.366,E2 -9743.366} C_VEL
LIN {X 0,Y 425.342,Z 597.499,A -85,B 0,C 180,E1 -9746.845,E2 -9746.845} C_VEL
LIN {X 0,Y 425.313,Z 597.503,A -85,B 0,C 180,E1 -9749.718,E2 -9749.718} C_VEL
LIN {X 0,Y 425.279,Z 597.506,A -85,B 0,C 180,E1 -9753.049,E2 -9753.049} C_VEL
LIN {X 0,Y 425.28,Z 597.508,A -85,B 0,C 180,E1 -9755.93,E2 -9755.93} C_VEL
LIN {X 0,Y 425.303,Z 597.505,A -85,B 0,C 180,E1 -9759.046,E2 -9759.046} C_VEL
LIN {X 0,Y 425.312,Z 597.506,A -85,B 0,C 180,E1 -9761.963,E2 -9761.963} C_VEL
LIN {X 0,Y 425.283,Z 597.513,A -85,B 0,C 180,E1 -9765.284,E2 -9765.284} C_VEL
LIN {X 0,Y 425.302,Z 597.505,A -85,B 0,C 180,E1 -9768.626,E2 -9768.626} C_VEL
LIN {X 0,Y 425.322,Z 597.506,A -85,B 0,C 180,E1 -9771.105,E2 -9771.105} C_VEL
LIN {X 0,Y 425.3,Z 597.506,A -85,B 0,C 180,E1 -9774.665,E2 -9774.665} C_VEL
LIN {X 0,Y 425.265,Z 597.512,A -85,B 0,C 180,E1 -9778.074,E2 -9778.074} C_VEL
LIN {X 0,Y 425.384,Z 597.636,A -85,B 0,C 180,E1 -9781.675,E2 -9781.675} C_VEL
LIN {X 0,Y 427.843,Z 609.233,A -85,B 0,C 180,E1 -9784.176,E2 -9784.176} C_VEL
LIN {X 0,Y 428.632,Z 614.617,A -85,B 0,C 180,E1 -9785.286,E2 -9785.286} C_VEL
LIN {X 0,Y 427.551,Z 630.473,A -85,B 0,C 180,E1 -9788.294,E2 -9788.294} C_VEL
LIN {X 0,Y 426.68,Z 646.075,A -85,B 0,C 180,E1 -9791.178,E2 -9791.178} C_VEL
LIN {X 0,Y 430.516,Z 672.071,A -85,B 0,C 180,E1 -9791.84,E2 -9791.84} C_VEL
LIN {X 0,Y 429.476,Z 755.495,A -85,B 0,C 180,E1 -9793.329,E2 -9793.329} C_VEL
LIN {X 0,Y 428.931,Z 769.137,A -85,B 0,C 180,E1 -9793.766,E2 -9793.766} C_VEL
LIN {X 0,Y 428.312,Z 781.51,A -85,B 0,C 180,E1 -9794.353,E2 -9794.353} C_VEL
LIN {X 0,Y 427.66,Z 793.416,A -85,B 0,C 180,E1 -9795.122,E2 -9795.122} C_VEL
LIN {X 0,Y 426.965,Z 804.747,A -85,B 0,C 180,E1 -9796.057,E2 -9796.057} C_VEL
LIN {X 0,Y 426.232,Z 815.266,A -85,B 0,C 180,E1 -9797.139,E2 -9797.139} C_VEL
LIN {X 0,Y 425.69,Z 824.595,A -85,B 0,C 180,E1 -9798.332,E2 -9798.332} C_VEL
LIN {X 0,Y 425.037,Z 833.676,A -85,B 0,C 180,E1 -9799.761,E2 -9799.761} C_VEL
LIN {X 0,Y 424.68,Z 841.009,A -85,B 0,C 180,E1 -9801.195,E2 -9801.195} C_VEL
LIN {X 0,Y 424.388,Z 845.962,A -85,B 0,C 180,E1 -9802.387,E2 -9802.387} C_VEL
LIN {X 0,Y 424.249,Z 850.403,A -85,B 0,C 180,E1 -9803.694,E2 -9803.694} C_VEL
LIN {X 0,Y 424.218,Z 854.477,A -85,B 0,C 180,E1 -9805.249,E2 -9805.249} C_VEL
LIN {X 0,Y 424.131,Z 856.378,A -85,B 0,C 180,E1 -9806.2,E2 -9806.2} C_VEL
LIN {X 0,Y 424.199,Z 857.81,A -85,B 0,C 180,E1 -9807.151,E2 -9807.151} C_VEL
LIN {X 0,Y 424.166,Z 858.833,A -85,B 0,C 180,E1 -9808.101,E2 -9808.101} C_VEL
LIN {X 0,Y 424.136,Z 859.461,A -85,B 0,C 180,E1 -9809.051,E2 -9809.051} C_VEL
LIN {X 0,Y 424.134,Z 859.682,A -85,B 0,C 180,E1 -9810,E2 -9810} C_VEL
LIN {X 0,Y 424.136,Z 859.461,A -85,B 0,C 180,E1 -9810.949,E2 -9810.949} C_VEL
LIN {X 0,Y 424.166,Z 858.847,A -85,B 0,C 180,E1 -9811.899,E2 -9811.899} C_VEL
LIN {X 0,Y 424.192,Z 857.837,A -85,B 0,C 180,E1 -9812.849,E2 -9812.849} C_VEL
LIN {X 0,Y 424.114,Z 856.396,A -85,B 0,C 180,E1 -9813.8,E2 -9813.8} C_VEL
LIN {X 0,Y 424.238,Z 853.405,A -85,B 0,C 180,E1 -9815.228,E2 -9815.228} C_VEL
LIN {X 0,Y 424.301,Z 849.34,A -85,B 0,C 180,E1 -9816.658,E2 -9816.658} C_VEL
LIN {X 0,Y 424.552,Z 843.078,A -85,B 0,C 180,E1 -9818.328,E2 -9818.328} C_VEL
LIN {X 0,Y 424.901,Z 836.252,A -85,B 0,C 180,E1 -9819.761,E2 -9819.761} C_VEL
LIN {X 0,Y 425.425,Z 827.767,A -85,B 0,C 180,E1 -9821.192,E2 -9821.192} C_VEL
LIN {X 0,Y 426.043,Z 819.023,A -85,B 0,C 180,E1 -9822.383,E2 -9822.383} C_VEL
LIN {X 0,Y 426.574,Z 809.066,A -85,B 0,C 180,E1 -9823.494,E2 -9823.494} C_VEL
LIN {X 0,Y 427.334,Z 797.553,A -85,B 0,C 180,E1 -9824.525,E2 -9824.525} C_VEL
LIN {X 0,Y 428.084,Z 785.594,A -85,B 0,C 180,E1 -9825.35,E2 -9825.35} C_VEL
LIN {X 0,Y 428.655,Z 773.173,A -85,B 0,C 180,E1 -9826,E2 -9826} C_VEL
LIN {X 0,Y 429.186,Z 760.422,A -85,B 0,C 180,E1 -9826.468,E2 -9826.468} C_VEL
LIN {X 0,Y 429.465,Z 747.094,A -85,B 0,C 180,E1 -9826.763,E2 -9826.763} C_VEL
LIN {X 0,Y 430.231,Z 671.564,A -85,B 0,C 180,E1 -9828.081,E2 -9828.081} C_VEL
LIN {X 0,Y 426.62,Z 646.858,A -85,B 0,C 180,E1 -9828.687,E2 -9828.687} C_VEL
LIN {X 0,Y 427.557,Z 630.606,A -85,B 0,C 180,E1 -9831.705,E2 -9831.705} C_VEL
LIN {X 0,Y 428.565,Z 615.944,A -85,B 0,C 180,E1 -9834.46,E2 -9834.46} C_VEL
LIN {X 0,Y 428.292,Z 611.904,A -85,B 0,C 180,E1 -9835.254,E2 -9835.254} C_VEL
LIN {X 0,Y 425.849,Z 599.69,A -85,B 0,C 180,E1 -9837.789,E2 -9837.789} C_VEL
LIN {X 0,Y 425.361,Z 597.503,A -85,B 0,C 180,E1 -9838.293,E2 -9838.293} C_VEL
LIN {X 0,Y 425.265,Z 597.513,A -85,B 0,C 180,E1 -9841.926,E2 -9841.926} C_VEL
LIN {X 0,Y 425.3,Z 597.503,A -85,B 0,C 180,E1 -9845.335,E2 -9845.335} C_VEL
LIN {X 0,Y 425.309,Z 597.504,A -85,B 0,C 180,E1 -9849.045,E2 -9849.045} C_VEL
LIN {X 0,Y 425.313,Z 597.503,A -85,B 0,C 180,E1 -9851.961,E2 -9851.961} C_VEL
LIN {X 0,Y 425.286,Z 597.506,A -85,B 0,C 180,E1 -9855.281,E2 -9855.281} C_VEL
LIN {X 0,Y 425.3,Z 597.51,A -85,B 0,C 180,E1 -9858.624,E2 -9858.624} C_VEL
LIN {X 0,Y 425.314,Z 597.505,A -85,B 0,C 180,E1 -9861.103,E2 -9861.103} C_VEL
LIN {X 0,Y 425.295,Z 597.51,A -85,B 0,C 180,E1 -9864.663,E2 -9864.663} C_VEL
LIN {X 0,Y 425.269,Z 597.507,A -85,B 0,C 180,E1 -9868.073,E2 -9868.073} C_VEL
LIN {X 0,Y 425.332,Z 597.502,A -85,B 0,C 180,E1 -9871.367,E2 -9871.367} C_VEL
LIN {X 0,Y 425.289,Z 597.507,A -85,B 0,C 180,E1 -9874.554,E2 -9874.554} C_VEL
LIN {X 0,Y 425.28,Z 597.507,A -85,B 0,C 180,E1 -9877.66,E2 -9877.66} C_VEL
LIN {X 0,Y 425.354,Z 597.499,A -85,B 0,C 180,E1 -9880.703,E2 -9880.703} C_VEL
LIN {X 0,Y 425.38,Z 597.495,A -85,B 0,C 180,E1 -9883.687,E2 -9883.687} C_VEL
LIN {X 0,Y 425.404,Z 597.493,A -85,B 0,C 180,E1 -9887.597,E2 -9887.597} C_VEL
LIN {X 0,Y 425.434,Z 597.492,A -85,B 0,C 180,E1 -9891.449,E2 -9891.449} C_VEL
LIN {X 0,Y 425.548,Z 597.472,A -85,B 0,C 180,E1 -9894.313,E2 -9894.313} C_VEL
LIN {X 0,Y 425.566,Z 597.471,A -85,B 0,C 180,E1 -9898.107,E2 -9898.107} C_VEL
LIN {X 0,Y 425.695,Z 597.456,A -85,B 0,C 180,E1 -9900,E2 -9900} C_VEL
LIN {X 0,Y 425.549,Z 597.473,A -85,B 0,C 180,E1 -9902.839,E2 -9902.839} C_VEL
LIN {X 0,Y 425.568,Z 597.476,A -85,B 0,C 180,E1 -9905.686,E2 -9905.686} C_VEL
LIN {X 0,Y 425.433,Z 597.487,A -85,B 0,C 180,E1 -9908.55,E2 -9908.55} C_VEL
LIN {X 0,Y 425.402,Z 597.491,A -85,B 0,C 180,E1 -9912.402,E2 -9912.402} C_VEL
LIN {X 0,Y 425.378,Z 597.495,A -85,B 0,C 180,E1 -9916.312,E2 -9916.312} C_VEL
LIN {X 0,Y 425.318,Z 597.506,A -85,B 0,C 180,E1 -9919.636,E2 -9919.636} C_VEL
LIN {X 0,Y 425.297,Z 597.505,A -85,B 0,C 180,E1 -9923.365,E2 -9923.365} C_VEL
LIN {X 0,Y 425.339,Z 597.498,A -85,B 0,C 180,E1 -9926.845,E2 -9926.845} C_VEL
LIN {X 0,Y 425.309,Z 597.506,A -85,B 0,C 180,E1 -9929.718,E2 -9929.718} C_VEL
LIN {X 0,Y 425.275,Z 597.506,A -85,B 0,C 180,E1 -9933.048,E2 -9933.048} C_VEL
LIN {X 0,Y 425.276,Z 597.512,A -85,B 0,C 180,E1 -9935.929,E2 -9935.929} C_VEL
LIN {X 0,Y 425.306,Z 597.502,A -85,B 0,C 180,E1 -9939.047,E2 -9939.047} C_VEL
LIN {X 0,Y 425.324,Z 597.503,A -85,B 0,C 180,E1 -9942.646,E2 -9942.646} C_VEL
LIN {X 0,Y 425.291,Z 597.504,A -85,B 0,C 180,E1 -9945.281,E2 -9945.281} C_VEL
LIN {X 0,Y 425.29,Z 597.508,A -85,B 0,C 180,E1 -9948.625,E2 -9948.625} C_VEL
LIN {X 0,Y 425.308,Z 597.503,A -85,B 0,C 180,E1 -9951.104,E2 -9951.104} C_VEL
LIN {X 0,Y 425.294,Z 597.509,A -85,B 0,C 180,E1 -9954.665,E2 -9954.665} C_VEL
LIN {X 0,Y 425.259,Z 597.511,A -85,B 0,C 180,E1 -9958.074,E2 -9958.074} C_VEL
LIN {X 0,Y 425.326,Z 597.5,A -85,B 0,C 180,E1 -9961.368,E2 -9961.368} C_VEL
LIN {X 0,Y 425.291,Z 597.511,A -85,B 0,C 180,E1 -9964.555,E2 -9964.555} C_VEL
LIN {X 0,Y 425.283,Z 597.505,A -85,B 0,C 180,E1 -9967.662,E2 -9967.662} C_VEL
LIN {X 0,Y 425.358,Z 597.504,A -85,B 0,C 180,E1 -9970.704,E2 -9970.704} C_VEL
LIN {X 0,Y 425.385,Z 597.493,A -85,B 0,C 180,E1 -9973.689,E2 -9973.689} C_VEL
LIN {X 0,Y 425.39,Z 597.496,A -85,B 0,C 180,E1 -9977.096,E2 -9977.096} C_VEL
LIN {X 0,Y 425.398,Z 597.494,A -85,B 0,C 180,E1 -9980.491,E2 -9980.491} C_VEL
LIN {X 0,Y 425.52,Z 597.479,A -85,B 0,C 180,E1 -9983.361,E2 -9983.361} C_VEL
LIN {X 0,Y 425.367,Z 597.499,A -85,B 0,C 180,E1 -9985.261,E2 -9985.261} C_VEL
LIN {X 0,Y 425.573,Z 597.469,A -85,B 0,C 180,E1 -9988.107,E2 -9988.107} C_VEL
LIN {X 0,Y 425.701,Z 597.453,A -85,B 0,C 180,E1 -9990,E2 -9990} C_VEL
LIN {X 0,Y 425.555,Z 597.476,A -85,B 0,C 180,E1 -9992.84,E2 -9992.84} C_VEL
LIN {X 0,Y 425.52,Z 597.477,A -85,B 0,C 180,E1 -9996.639,E2 -9996.639} C_VEL
LIN {X 0,Y 425.399,Z 597.492,A -85,B 0,C 180,E1 -9999.161,E2 -9999.161} C_VEL
LIN {X 0,Y 424.727,Z 597.58,A -85,B 0,C 180,E1 -9999.95,E2 -9999.95} C_VEL
LIN {X 0,Y 421.878,Z 597.937,A -85,B 0,C 180,E1 -10001.234,E2 -10001.234} C_VEL
LIN {X 0,Y 419.462,Z 598.235,A -85,B 0,C 180,E1 -10002.27,E2 -10002.27} C_VEL
LIN {X 0,Y 418.411,Z 598.366,A -85,B 0,C 180,E1 -10003.071,E2 -10003.071} C_VEL
LIN {X 0,Y 418.319,Z 598.376,A -85,B 0,C 180,E1 -10003.342,E2 -10003.342} C_VEL
LIN {X 0,Y 418.309,Z 598.375,A -85,B 0,C 180,E1 -10006.735,E2 -10006.735} C_VEL
LIN {X 0,Y 418.267,Z 598.385,A -85,B 0,C 180,E1 -10009.79,E2 -10009.79} C_VEL
LIN {X 0,Y 418.298,Z 598.384,A -85,B 0,C 180,E1 -10013.452,E2 -10013.452} C_VEL
LIN {X 0,Y 419.888,Z 607.352,A -85,B 0,C 180,E1 -10015.796,E2 -10015.796} C_VEL
LIN {X 0,Y 419.864,Z 608.576,A -85,B 0,C 180,E1 -10016.098,E2 -10016.098} C_VEL
LIN {X 0,Y 423.815,Z 627.203,A -85,B 0,C 180,E1 -10016.631,E2 -10016.631} C_VEL
LIN {X 0,Y 422.634,Z 715.385,A -85,B 0,C 180,E1 -10018.215,E2 -10018.215} C_VEL
LIN {X 0,Y 422.251,Z 728.923,A -85,B 0,C 180,E1 -10018.654,E2 -10018.654} C_VEL
LIN {X 0,Y 421.851,Z 740.947,A -85,B 0,C 180,E1 -10019.231,E2 -10019.231} C_VEL
LIN {X 0,Y 421.248,Z 752.072,A -85,B 0,C 180,E1 -10019.937,E2 -10019.937} C_VEL
LIN {X 0,Y 420.53,Z 764.023,A -85,B 0,C 180,E1 -10020.923,E2 -10020.923} C_VEL
LIN {X 0,Y 419.84,Z 774.586,A -85,B 0,C 180,E1 -10022.02,E2 -10022.02} C_VEL
LIN {X 0,Y 419.214,Z 784.378,A -85,B 0,C 180,E1 -10023.289,E2 -10023.289} C_VEL
LIN {X 0,Y 418.571,Z 792.819,A -85,B 0,C 180,E1 -10024.642,E2 -10024.642} C_VEL
LIN {X 0,Y 418.026,Z 800.629,A -85,B 0,C 180,E1 -10026.198,E2 -10026.198} C_VEL
LIN {X 0,Y 417.677,Z 806.67,A -85,B 0,C 180,E1 -10027.737,E2 -10027.737} C_VEL
LIN {X 0,Y 417.383,Z 811.255,A -85,B 0,C 180,E1 -10029.236,E2 -10029.236} C_VEL
LIN {X 0,Y 417.154,Z 815.325,A -85,B 0,C 180,E1 -10031.074,E2 -10031.074} C_VEL
LIN {X 0,Y 417.018,Z 817.254,A -85,B 0,C 180,E1 -10032.384,E2 -10032.384} C_VEL
LIN {X 0,Y 416.965,Z 818.455,A -85,B 0,C 180,E1 -10033.713,E2 -10033.713} C_VEL
LIN {X 0,Y 416.928,Z 818.907,A -85,B 0,C 180,E1 -10035.069,E2 -10035.069} C_VEL
LIN {X 0,Y 416.977,Z 818.524,A -85,B 0,C 180,E1 -10036.447,E2 -10036.447} C_VEL
LIN {X 0,Y 417.039,Z 817.299,A -85,B 0,C 180,E1 -10037.857,E2 -10037.857} C_VEL
LIN {X 0,Y 417.198,Z 815.161,A -85,B 0,C 180,E1 -10039.291,E2 -10039.291} C_VEL
LIN {X 0,Y 417.413,Z 811.989,A -85,B 0,C 180,E1 -10040.758,E2 -10040.758} C_VEL
LIN {X 0,Y 417.704,Z 807.626,A -85,B 0,C 180,E1 -10042.258,E2 -10042.258} C_VEL
LIN {X 0,Y 418.154,Z 801.121,A -85,B 0,C 180,E1 -10043.968,E2 -10043.968} C_VEL
LIN {X 0,Y 418.615,Z 794.412,A -85,B 0,C 180,E1 -10045.349,E2 -10045.349} C_VEL
LIN {X 0,Y 419.238,Z 786.269,A -85,B 0,C 180,E1 -10046.705,E2 -10046.705} C_VEL
LIN {X 0,Y 419.933,Z 776.85,A -85,B 0,C 180,E1 -10047.981,E2 -10047.981} C_VEL
LIN {X 0,Y 420.663,Z 766.722,A -85,B 0,C 180,E1 -10049.087,E2 -10049.087} C_VEL
LIN {X 0,Y 421.372,Z 755.619,A -85,B 0,C 180,E1 -10050.053,E2 -10050.053} C_VEL
LIN {X 0,Y 421.967,Z 744.031,A -85,B 0,C 180,E1 -10050.846,E2 -10050.846} C_VEL
LIN {X 0,Y 422.532,Z 731.922,A -85,B 0,C 180,E1 -10051.469,E2 -10051.469} C_VEL
LIN {X 0,Y 422.845,Z 719.959,A -85,B 0,C 180,E1 -10051.903,E2 -10051.903} C_VEL
LIN {X 0,Y 423.147,Z 702.876,A -85,B 0,C 180,E1 -10052.266,E2 -10052.266} C_VEL
LIN {X 0,Y 424.268,Z 627.825,A -85,B 0,C 180,E1 -10053.619,E2 -10053.619} C_VEL
LIN {X 0,Y 420.253,Z 609.784,A -85,B 0,C 180,E1 -10054.188,E2 -10054.188} C_VEL
LIN {X 0,Y 419.754,Z 605.756,A -85,B 0,C 180,E1 -10055.256,E2 -10055.256} C_VEL
LIN {X 0,Y 418.261,Z 598.386,A -85,B 0,C 180,E1 -10057.315,E2 -10057.315} C_VEL
LIN {X 0,Y 418.273,Z 598.385,A -85,B 0,C 180,E1 -10060.364,E2 -10060.364} C_VEL
LIN {X 0,Y 418.307,Z 598.378,A -85,B 0,C 180,E1 -10063.405,E2 -10063.405} C_VEL
LIN {X 0,Y 418.346,Z 598.375,A -85,B 0,C 180,E1 -10066.994,E2 -10066.994} C_VEL
LIN {X 0,Y 418.351,Z 598.375,A -85,B 0,C 180,E1 -10070.329,E2 -10070.329} C_VEL
LIN {X 0,Y 418.486,Z 598.357,A -85,B 0,C 180,E1 -10073.249,E2 -10073.249} C_VEL
LIN {X 0,Y 418.34,Z 598.376,A -85,B 0,C 180,E1 -10075.182,E2 -10075.182} C_VEL
LIN {X 0,Y 418.537,Z 598.348,A -85,B 0,C 180,E1 -10078.076,E2 -10078.076} C_VEL
LIN {X 0,Y 418.665,Z 598.332,A -85,B 0,C 180,E1 -10080,E2 -10080} C_VEL
LIN {X 0,Y 418.504,Z 598.357,A -85,B 0,C 180,E1 -10082.888,E2 -10082.888} C_VEL
LIN {X 0,Y 418.526,Z 598.349,A -85,B 0,C 180,E1 -10085.783,E2 -10085.783} C_VEL
LIN {X 0,Y 418.392,Z 598.37,A -85,B 0,C 180,E1 -10088.696,E2 -10088.696} C_VEL
LIN {X 0,Y 418.326,Z 598.374,A -85,B 0,C 180,E1 -10091.631,E2 -10091.631} C_VEL
LIN {X 0,Y 418.299,Z 598.379,A -85,B 0,C 180,E1 -10094.598,E2 -10094.598} C_VEL
LIN {X 0,Y 418.28,Z 598.381,A -85,B 0,C 180,E1 -10097.605,E2 -10097.605} C_VEL
LIN {X 0,Y 418.242,Z 598.385,A -85,B 0,C 180,E1 -10100.664,E2 -10100.664} C_VEL
LIN {X 0,Y 418.281,Z 598.38,A -85,B 0,C 180,E1 -10103.782,E2 -10103.782} C_VEL
LIN {X 0,Y 418.304,Z 598.378,A -85,B 0,C 180,E1 -10107.071,E2 -10107.071} C_VEL
LIN {X 0,Y 418.258,Z 598.38,A -85,B 0,C 180,E1 -10110.272,E2 -10110.272} C_VEL
LIN {X 0,Y 418.244,Z 598.384,A -85,B 0,C 180,E1 -10113.678,E2 -10113.678} C_VEL
LIN {X 0,Y 418.242,Z 598.388,A -85,B 0,C 180,E1 -10117.225,E2 -10117.225} C_VEL
LIN {X 0,Y 418.258,Z 598.385,A -85,B 0,C 180,E1 -10119.682,E2 -10119.682} C_VEL
LIN {X 0,Y 418.244,Z 598.385,A -85,B 0,C 180,E1 -10122.325,E2 -10122.325} C_VEL
LIN {X 0,Y 418.235,Z 598.389,A -85,B 0,C 180,E1 -10125.11,E2 -10125.11} C_VEL
LIN {X 0,Y 418.254,Z 598.386,A -85,B 0,C 180,E1 -10127.77,E2 -10127.77} C_VEL
LIN {X 0,Y 418.266,Z 598.382,A -85,B 0,C 180,E1 -10130.618,E2 -10130.618} C_VEL
LIN {X 0,Y 418.246,Z 598.388,A -85,B 0,C 180,E1 -10133.977,E2 -10133.977} C_VEL
LIN {X 0,Y 418.257,Z 598.389,A -85,B 0,C 180,E1 -10137.157,E2 -10137.157} C_VEL
LIN {X 0,Y 418.269,Z 598.385,A -85,B 0,C 180,E1 -10140.896,E2 -10140.896} C_VEL
LIN {X 0,Y 418.316,Z 598.508,A -85,B 0,C 180,E1 -10141.362,E2 -10141.362} C_VEL
LIN {X 0,Y 420.902,Z 610.49,A -85,B 0,C 180,E1 -10144.005,E2 -10144.005} C_VEL
LIN {X 0,Y 421.719,Z 615.774,A -85,B 0,C 180,E1 -10145.116,E2 -10145.116} C_VEL
LIN {X 0,Y 420.783,Z 628.922,A -85,B 0,C 180,E1 -10147.668,E2 -10147.668} C_VEL
LIN {X 0,Y 419.772,Z 645.442,A -85,B 0,C 180,E1 -10150.819,E2 -10150.819} C_VEL
LIN {X 0,Y 423.814,Z 672.774,A -85,B 0,C 180,E1 -10151.542,E2 -10151.542} C_VEL
LIN {X 0,Y 422.782,Z 754.342,A -85,B 0,C 180,E1 -10153.026,E2 -10153.026} C_VEL
LIN {X 0,Y 422.217,Z 767.473,A -85,B 0,C 180,E1 -10153.438,E2 -10153.438} C_VEL
LIN {X 0,Y 421.563,Z 780.194,A -85,B 0,C 180,E1 -10154.034,E2 -10154.034} C_VEL
LIN {X 0,Y 420.885,Z 791.563,A -85,B 0,C 180,E1 -10154.753,E2 -10154.753} C_VEL
LIN {X 0,Y 420.118,Z 803.522,A -85,B 0,C 180,E1 -10155.735,E2 -10155.735} C_VEL
LIN {X 0,Y 419.414,Z 813.908,A -85,B 0,C 180,E1 -10156.803,E2 -10156.803} C_VEL
LIN {X 0,Y 418.817,Z 822.58,A -85,B 0,C 180,E1 -10157.892,E2 -10157.892} C_VEL
LIN {X 0,Y 418.212,Z 830.587,A -85,B 0,C 180,E1 -10159.103,E2 -10159.103} C_VEL
LIN {X 0,Y 417.729,Z 838.418,A -85,B 0,C 180,E1 -10160.559,E2 -10160.559} C_VEL
LIN {X 0,Y 417.336,Z 845.639,A -85,B 0,C 180,E1 -10162.258,E2 -10162.258} C_VEL
LIN {X 0,Y 417.175,Z 850.409,A -85,B 0,C 180,E1 -10163.698,E2 -10163.698} C_VEL
LIN {X 0,Y 417.148,Z 854.143,A -85,B 0,C 180,E1 -10165.168,E2 -10165.168} C_VEL
LIN {X 0,Y 417.045,Z 856.04,A -85,B 0,C 180,E1 -10166.135,E2 -10166.135} C_VEL
LIN {X 0,Y 417.097,Z 857.47,A -85,B 0,C 180,E1 -10167.103,E2 -10167.103} C_VEL
LIN {X 0,Y 417.093,Z 858.494,A -85,B 0,C 180,E1 -10168.069,E2 -10168.069} C_VEL
LIN {X 0,Y 417.056,Z 859.12,A -85,B 0,C 180,E1 -10169.034,E2 -10169.034} C_VEL
LIN {X 0,Y 417.051,Z 859.336,A -85,B 0,C 180,E1 -10170,E2 -10170} C_VEL
LIN {X 0,Y 417.056,Z 859.113,A -85,B 0,C 180,E1 -10170.966,E2 -10170.966} C_VEL
LIN {X 0,Y 417.092,Z 858.497,A -85,B 0,C 180,E1 -10171.931,E2 -10171.931} C_VEL
LIN {X 0,Y 417.089,Z 857.481,A -85,B 0,C 180,E1 -10172.897,E2 -10172.897} C_VEL
LIN {X 0,Y 417.029,Z 856.033,A -85,B 0,C 180,E1 -10173.865,E2 -10173.865} C_VEL
LIN {X 0,Y 417.149,Z 853.032,A -85,B 0,C 180,E1 -10175.317,E2 -10175.317} C_VEL
LIN {X 0,Y 417.233,Z 848.956,A -85,B 0,C 180,E1 -10176.771,E2 -10176.771} C_VEL
LIN {X 0,Y 417.508,Z 842.679,A -85,B 0,C 180,E1 -10178.47,E2 -10178.47} C_VEL
LIN {X 0,Y 417.877,Z 835.835,A -85,B 0,C 180,E1 -10179.926,E2 -10179.926} C_VEL
LIN {X 0,Y 418.43,Z 827.315,A -85,B 0,C 180,E1 -10181.382,E2 -10181.382} C_VEL
LIN {X 0,Y 419.051,Z 818.534,A -85,B 0,C 180,E1 -10182.593,E2 -10182.593} C_VEL
LIN {X 0,Y 419.706,Z 807.962,A -85,B 0,C 180,E1 -10183.78,E2 -10183.78} C_VEL
LIN {X 0,Y 420.434,Z 796.961,A -85,B 0,C 180,E1 -10184.768,E2 -10184.768} C_VEL
LIN {X 0,Y 421.209,Z 784.906,A -85,B 0,C 180,E1 -10185.607,E2 -10185.607} C_VEL
